// ---- XTS/Xpu/fb_Xpu.TcPOU
//---------------------------------------------------------------------------------------------------------------
//
//  HAUD 2023.12.14
//
//  - XTS_TRANSPORT_LAYER
//
//  fb_Xpu
//  - connect XTS_Utility.lib to TcCom
//  - cyclic plausibility checks
//  - cyclic ModuleInfoData
//
//  - connection to TcCom Server for local FB instances
//
//
//  CTRL / STATE --> see proprerties
//  structs for use of function block via mapping
//  cyclic check for new command
//
//  VAR INPUT / OUTPUT --> see properties
//
//---------------------------------------------------------------------------------------------------------------
// This SOFTWARE is provided as an Exemple by THE PROVIDER "as is" and "with all faults." THE PROVIDER makes no 
// representations or warranties of any kind concerning the safety, suitability, lack of viruses, inaccuracies, 
// typographical errors, or other harmful components of this SOFTWARE. There are inherent dangers in the use of 
// any software, and you are solely responsible for determining whether this SOFTWARE is compatible with your 
// equipment and other software installed on your equipment. You are also solely responsible for the protection 
// of your equipment and backup of your data, and THE PROVIDER will not be liable for any damages you may suffer 
// in connection with using, modifying, or distributing this SOFTWARE.
//---------------------------------------------------------------------------------------------------------------
FUNCTION_BLOCK fb_Xpu //IMPLEMENTS I_Xpu
VAR
  _eCheck                     : E_XPU_CHECK;
  _eInit                      : E_XPU_INIT;       // MUST equal INIT_DONE for anything to work
  _sVersionXpu                : STRING(80);       // only valid after successful init
  _sVersionNctController      : STRING(80);       // only valid afetr successful init
  //-------------------------------------------------------------------------------------------------
  // XTS Environment; ProcessingUnit, Part, Track, Mover
  //  - instances are initialized by getting OTCIDs
  //-------------------------------------------------------------------------------------------------
  _nXpu                       : UINT := 1;  // input property in case of multiple XPU in project
  _nGroup                     : UINT;       // input property in case of multiple Xpu in project

  _nTrack                     : UINT := 1;  // this example is intended for one track only

  {attribute 'displaymode':='hex'}
  _CaGroupOID                 : OTCID; // input property frome cyclic CA group interface, MUST be set in order to do successful INIT

  // checked and evaluated in XpuCheckCycle()
  _bAllPositionsValid,
  _bMoverIdDetectionValid,
  _bMoverIdDetectionError     : BOOL;

  _nDetectedMoverCount,
  _nExpectedMoverCount        : UINT;

  _XpuOperationMode           : OperationMode;
  _MoverIdDetectionMode       : MoverIdDetectionMode;

  // XTS_Utility connection to TcCOM Object
  _fbEnvironment              : Tc3_XTS_Utility.FB_TcIoXtsEnvironment;

  // local instances of members of Environment
  // local members are connected to TcCOM by XpuInit()
  _fbProcessingUnit           : Tc3_XTS_Utility.FB_TcIoXtsProcessingUnit;

  _fbXpuPart                  : Tc3_XTS_Utility.FB_TcIoXtsXpuPart;
  _fbXpuTrack                 : Tc3_XTS_Utility.FB_TcIoXtsXpuTrack;

  _fbMc2CaGroup               : Tc3_XTS_Utility.FB_Mc2CaGroup;

  _fbPartModules              : ARRAY[1..MAX_MODULE]  OF Tc3_XTS_Utility.FB_TcIoXtsPartModule;
  _fbMoverXpu                 : ARRAY[1..MAX_MOVER]   OF Tc3_XTS_Utility.FB_TcIoXtsXpuMover;

  _fbParameterSet             : ARRAY[1..MAX_PARAMETER_SET] OF Tc3_XTS_Utility.FB_TcIoXtsParameterSet;

  _fbNctController            : Tc3_XTS_Utility.FB_TcIoXtsNctController;

  _ItfNctBaseUnit              : ARRAY[1..MAX_NCT_BASE_UNIT] OF Tc3_XTS_Utility.I_TcIoXtsNctBaseUnitInterface;


  // TcCOM ObjectId (who am I talking to?)
  {attribute 'displaymode':='hex'}
  _Xpu_OTCID                  : OTCID;
  {attribute 'displaymode':='hex'}
  _Nct_OTCID                  : OTCID;
  {attribute 'displaymode':='hex'}
  _Group_OTCID                : ARRAY[1..MAX_GROUP]         OF OTCID; // OTCID read from XPU
  {attribute 'displaymode':='hex'}
  _Part_OTCID                 : ARRAY[1..MAX_PART]          OF OTCID;
  {attribute 'displaymode':='hex'}
  _Track_OTCID                : ARRAY[1..MAX_TRACK]         OF OTCID;
  {attribute 'displaymode':='hex'}
  _Mov_OTCID                  : ARRAY[1..MAX_MOVER]         OF OTCID;
  {attribute 'displaymode':='hex'}
  _Module_OTCID               : ARRAY[1..MAX_MODULE]        OF OTCID;
  {attribute 'displaymode':='hex'}
  _ParameterSet_OTCID         : ARRAY[1..MAX_PARAMETER_SET] OF OTCID;
  {attribute 'displaymode':='hex'}
  _NctBaseUnit_OTCID          : ARRAY[1..MAX_NCT_BASE_UNIT] OF OTCID;

  // COE Data access
  _ModuleInfoData             : REFERENCE TO ARRAY[1..MAX_MODULE] OF Tc3_XTS_Utility.ST_InfoDataView;
  _bModulePower               : ARRAY[1..MAX_MODULE] OF BOOL;

  // double check RailLength, XpuInit() will get stuck in error if not configured correctly
  _RailLengthXpu              : LREAL;
  _RailLengthGroup            : LREAL;

  _nLengthXpu,
  _nLengthGroup               : UINT;

  _nNctBaseUnitCount,
  _nParameterSetCount,
  _nInfoServerCount,
  _nIfoStationCount,
  _nPartCount,
  _nTrackCount,
  _nTaskCount,
  _nMoverCount,
  _nModuleCount               : UINT;

  _ix                         : UINT;

  {attribute 'hide'}
  _XpuInfo                    : ST_XPU_INFO;

  _stMsg                      : ST_Message;
  _eMessageLevel              : E_MessageType;
END_VAR

// get DcLink information from motor modules
PROPERTY AllModulesDcLink : bool
GET
VAR
  _bTmp     : BOOL;
  _nModule  : UINT;
END_VAR
IF NOT (_eInit = E_XPU_INIT.INIT_DONE) THEN RETURN; END_IF

FOR _nModule := 1 TO _nModuleCount
DO
  IF NOT _bModulePower[_nModule] // information comes from cyclic call in Cycle(): ModuleInfoData()
  THEN
    _bTmp  := FALSE;
    EXIT;
  ELSE
    _bTmp  := TRUE;
  END_IF
END_FOR

AllModulesDcLink := _bTmp;
END_GET
END_PROPERTY

PROPERTY CaGroupOID : OTCID
SET
// Group OTCID must come from the CA Group mapping in NC.Objects
_CaGroupOID := CaGroupOID;
END_SET
END_PROPERTY

METHOD Cycle : E_PROGRESS
VAR_INPUT
  Enable      : BOOL; // enable to do cyclic checks on Environment and its members
END_VAR
VAR_IN_OUT
  _eChk       : E_XPU_CHECK;
END_VAR
VAR_INST

  _eJobResult,
  _eResult      : E_PROGRESS;
  _eState       : E_PROGRESS := E_PROGRESS.PROGRESS_INIT;

END_VAR
IF NOT Enable
THEN
  ModuleInfoData(FALSE);

  _eResult  :=
  _eState   := E_PROGRESS.PROGRESS_INIT; 
  _eChk     := E_XPU_CHECK.INIT_CHECK;
END_IF 
//-----------------------------------------------------------------------------
// cyclic data fetch from Environment, ProcessingUnit, Part, ...
//-----------------------------------------------------------------------------
CASE _eState
OF
  E_PROGRESS.PROGRESS_INIT:
    IF Enable
    THEN
      _eState := _eResult         := E_PROGRESS.PROGRESS_BUSY;
    END_IF

  //---------------------------------------------------------------------------
  E_PROGRESS.PROGRESS_BUSY:       // get data from Xpu, ProcessingUnit, Part, XpuCaGroup
    _eState                       := E_PROGRESS.PROGRESS_STARTUP;

    _bAllPositionsValid           := _fbProcessingUnit.GetAreAllPositionsValid();
    _nDetectedMoverCount          := TO_UINT(_fbProcessingUnit.GetDetectedMoverCount());
    _nExpectedMoverCount          := TO_UINT(_fbProcessingUnit.GetExpectedMoverCount());
  
    _XpuOperationMode             := _fbProcessingUnit.GetOperationMode();
    _MoverIdDetectionMode         := _fbProcessingUnit.GetMoverIdDetectionMode();
  
    _RailLengthXpu                := _fbXpuPart.GetLength();
    _RailLengthGroup              := _fbMc2CaGroup.GetRailLength();
    _nLengthXpu                   := TO_UINT(_RailLengthXpu);
    _nLengthGroup                 := TO_UINT(_RailLengthGroup);
END_CASE
//-----------------------------------------------------------------------------
//-----------------------------------------------------------------------------
CASE _eState
OF
  //---------------------------------------------------------------------------
  E_PROGRESS.PROGRESS_STARTUP:    // check data for errors
    IF NOT (_bAllPositionsValid)
    THEN
      _eChk                       := E_XPU_CHECK.PROCESSING_UNIT_POSITIONS_VALID;
      _eState := _eResult         := E_PROGRESS.PROGRESS_ERROR;

      _stMsg.eType                := E_MessageType.eMessageError;
      _stMsg.eSubdevice           := e_Subdevice.Xpu_fbProcessingUnit;
      _stMsg.iErrorNumber         := 0;
      _stMsg.sText                := concat(TO_STRING(E_XPU_CHECK.PROCESSING_UNIT_POSITIONS_VALID), ': ');
      _stMsg.sText                := concat(_stMsg.sText, TO_STRING(_eResult));
      f_MessageSet(_stMsg);

    ELSIF NOT (_nLengthXpu > 0)
    THEN
      _eChk                       := E_XPU_CHECK.XPU_RAIL_LENGTH;
      _eState := _eResult         := E_PROGRESS.PROGRESS_ERROR;

      _stMsg.eType                := E_MessageType.eMessageError;
      _stMsg.eSubdevice           := e_Subdevice.Xpu_fbProcessingUnit;
      _stMsg.iErrorNumber         := 0;
      _stMsg.sText                := concat(TO_STRING(E_XPU_CHECK.XPU_RAIL_LENGTH), ': ');
      _stMsg.sText                := concat(_stMsg.sText, TO_STRING(_eResult));
      f_MessageSet(_stMsg);

    ELSIF NOT (_nLengthGroup > 0)
    THEN
      _eChk                       := E_XPU_CHECK.GROUP_RAIL_LENGTH;
      _eState := _eResult         := E_PROGRESS.PROGRESS_ERROR;
     
      _stMsg.eType                := E_MessageType.eMessageError;
      _stMsg.eSubdevice           := e_Subdevice.Xpu_fbProcessingUnit;
      _stMsg.iErrorNumber         := 0;
      _stMsg.sText                := concat(TO_STRING(E_XPU_CHECK.GROUP_RAIL_LENGTH), ': ');
      _stMsg.sText                := concat(_stMsg.sText, TO_STRING(_eResult));
      f_MessageSet(_stMsg);

    ELSIF NOT (_nDetectedMoverCount = _nExpectedMoverCount)
    THEN
      _bMoverIdDetectionValid     := FALSE;
      _eChk                       := E_XPU_CHECK.MOVER_COUNT_NOT_EQUAL;
      _eState := _eResult         := E_PROGRESS.PROGRESS_ERROR;

      _stMsg.eType                := E_MessageType.eMessageError;
      _stMsg.eSubdevice           := e_Subdevice.Xpu_fbProcessingUnit;
      _stMsg.iErrorNumber         := 0;
      _stMsg.sText                := concat(TO_STRING(E_XPU_CHECK.MOVER_COUNT_NOT_EQUAL), ': ');
      _stMsg.sText                := concat(_stMsg.sText, TO_STRING(_eResult));
      f_MessageSet(_stMsg);
  
    ELSIF NOT (_nLengthXpu = _nLengthGroup)
    THEN
      _eChk                       := E_XPU_CHECK.RAIL_LENGTH_COMPARE;
      _eState := _eResult         := E_PROGRESS.PROGRESS_ERROR;
 
      _stMsg.eType                := E_MessageType.eMessageError;
      _stMsg.eSubdevice           := e_Subdevice.Xpu_fbProcessingUnit;
      _stMsg.iErrorNumber         := 0;
      _stMsg.sText                := concat(TO_STRING(E_XPU_CHECK.RAIL_LENGTH_COMPARE), ': ');
      _stMsg.sText                := concat(_stMsg.sText, TO_STRING(_eResult));
      f_MessageSet(_stMsg);

    ELSE
      _eResult                    := E_PROGRESS.PROGRESS_WORKING;

      IF NOT (__ISVALIDREF(_ModuleInfoData))
      THEN
        _eState                   := E_PROGRESS.PROGRESS_BUSY;

        _stMsg.eType              := E_MessageType.eMessageError;
        _stMsg.eSubdevice         := e_Subdevice.Xpu_fbPartModules;
        _stMsg.iErrorNumber       := 0;
        _stMsg.sText              := concat(TO_STRING(_eState), ': ');
        _stMsg.sText              := concat(_stMsg.sText, 'NOT VALID _ModuleInfoData ref');
      ELSE
        _eJobResult               := ModuleInfoData(TRUE);
  
        IF (_eJobResult = E_PROGRESS.PROGRESS_DONE)
        THEN
          _eState                 := E_PROGRESS.PROGRESS_BUSY;
        END_IF  
      END_IF
    END_IF
END_CASE

Cycle                             := _eResult;
END_METHOD

METHOD GetEnvironment : I_TcIoXtsEnvironment
VAR_INPUT
END_VAR
IF NOT (_eInit = E_XPU_INIT.INIT_DONE) THEN RETURN; END_IF

GetEnvironment := _fbEnvironment;
END_METHOD

METHOD GetNctBaseUnit : Tc3_XTS_Utility.I_TcIoXtsNctBaseUnitInterface
VAR_INPUT
  Index     : UINT;
END_VAR
IF NOT (_eInit = E_XPU_INIT.INIT_DONE) THEN RETURN; END_IF

IF NOT (Index > 0) OR
   NOT (Index < MAX_NCT_BASE_UNIT+1)
THEN
  RETURN;
ELSE
  GetNctBaseUnit    := _ItfNctBaseUnit[Index];
END_IF
END_METHOD

METHOD GetNctController : Tc3_XTS_Utility.I_TcIoXtsNctController
VAR_INPUT
END_VAR
IF NOT (_eInit = E_XPU_INIT.INIT_DONE) THEN RETURN; END_IF

GetNctController := _fbNctController;
END_METHOD

METHOD GetParameterSet : I_TcIoXtsParameterSet
VAR_INPUT
  Index     : UINT;
END_VAR
IF NOT (_eInit = E_XPU_INIT.INIT_DONE) THEN RETURN; END_IF

IF NOT (Index > 0) OR
   NOT (Index < MAX_PARAMETER_SET+1)
THEN
  RETURN;
ELSE
  GetParameterSet   := _fbParameterSet[Index];
END_IF
END_METHOD

METHOD GetProcessingUnit : Tc3_XTS_Utility.I_TcIoXtsProcessingUnit
VAR_INPUT
END_VAR
IF NOT (_eInit = E_XPU_INIT.INIT_DONE) THEN RETURN; END_IF

GetProcessingUnit := _fbProcessingUnit;
END_METHOD

METHOD GetXpuMover : Tc3_XTS_Utility.I_TcIoXtsXpuMover
VAR_INPUT
  Index     : UINT;
END_VAR
IF NOT (_eInit = E_XPU_INIT.INIT_DONE) THEN RETURN; END_IF

IF NOT (Index > 0) OR
   NOT (Index < MAX_MOVER+1)
THEN
  RETURN;
ELSE
  GetXpuMover   := _fbMoverXpu[Index];
END_IF
END_METHOD

// mothers' little helper for display in visu
METHOD IdDetectionModeToString : string(20)
VAR
  _DetectionMode    : MoverIdDetectionMode; // Mover ID detection procedure
END_VAR
// just a little helper for visu display
IF NOT (_eInit = E_XPU_INIT.INIT_DONE) THEN IdDetectionModeToString := 'INIT required'; RETURN; END_IF

_DetectionMode := _fbProcessingUnit.GetMoverIdDetectionMode();

CASE _DetectionMode
OF
  MoverIdDetectionMode.Standard:
    IdDetectionModeToString       := 'Standard';

  MoverIdDetectionMode.Mover1:
    IdDetectionModeToString       := 'Mover 1';

  MoverIdDetectionMode.MultipleMover1:
    IdDetectionModeToString       := 'Multiple Mover 1';

ELSE
    IdDetectionModeToString       := 'UNKNOWN Mode';
END_CASE
END_METHOD

PROPERTY MessageLevel : e_messagetype
SET
_eMessageLevel := MessageLevel;
END_SET
END_PROPERTY

// mothers' little helper for display in visu
METHOD PRIVATE ModuleInfoData : E_PROGRESS
VAR_INPUT
  Enable        : BOOL; // enable to read ST_InfoDataView for diag/display
END_VAR
VAR_INST
  _idt,
  _nModule : UINT;
  _eReturn,
  _eState       : E_PROGRESS;
  _aPcbTemp     : ARRAY[1..4] OF REAL;
END_VAR
//---------------------------------------------------------------------------------------------
// just a little helper for visu display
// collects module data for local data
//---------------------------------------------------------------------------------------------
IF NOT (_eInit = E_XPU_INIT.INIT_DONE)      // if Xpu init is not done, just leave
THEN 
  RETURN; 
END_IF
//---------------------------------------------------------------------------------------------
IF NOT Enable                               // clear states on request
THEN
  _eReturn                                  := 
  _eState                                   := E_PROGRESS.PROGRESS_INIT; 
END_IF 
//---------------------------------------------------------------------------------------------
IF NOT (__ISVALIDREF(_ModuleInfoData))      // datafield not connected, error and leave
THEN
  ModuleInfoData                            := E_PROGRESS.PROGRESS_ERROR;
  RETURN;
END_IF
//---------------------------------------------------------------------------------------------
CASE _eState                                // get InfoData from motor modules
OF
  //-------------------------------------------------------------------------------------------
  E_PROGRESS.PROGRESS_INIT:
    IF Enable
    THEN
      _eState                                             := E_PROGRESS.PROGRESS_BUSY;
      _nModule                                            := 1;
    END_IF
END_CASE
CASE _eState
OF
  //-------------------------------------------------------------------------------------------
  E_PROGRESS.PROGRESS_BUSY:
    _eState                                               := E_PROGRESS.PROGRESS_PREPARE;

    _ModuleInfoData[_nModule].fAuxiliaryVoltage_5V        := _fbPartModules[_nModule].GetAuxiliaryVoltage5V();
    _ModuleInfoData[_nModule].fAuxiliaryVoltage_10V       := _fbPartModules[_nModule].GetAuxiliaryVoltage10V();
    _ModuleInfoData[_nModule].fAuxiliaryVoltage_24V       := _fbPartModules[_nModule].GetAuxiliaryVoltage24V();

    _ModuleInfoData[_nModule].fDcLinkVoltage              := _fbPartModules[_nModule].GetDCLinkVoltage();

    IF (_ModuleInfoData[_nModule].fDcLinkVoltage > 48.0*0.85) AND
       (_ModuleInfoData[_nModule].fDcLinkVoltage < 48.0*1.15)
    THEN
      _bModulePower[_nModule]                             := TRUE;
    ELSE
      _bModulePower[_nModule]                             := SEL((_XpuOperationMode = OperationMode.Simulation), FALSE, TRUE);
    END_IF

    _ModuleInfoData[_nModule].nCurrentScaling             := TO_INT(_fbPartModules[_nModule].GetCurrentScaling());

    _ModuleInfoData[_nModule].nDeviceInfo                 := _fbPartModules[_nModule].GetDeviceInfo();

    IF (_XpuOperationMode = OperationMode.Normal)
    THEN
      _ModuleInfoData[_nModule].fAverageTemp              := 0.0;
  
      _aPcbTemp                                           := _fbPartModules[_nModule].GetPCBTemperatures();
  
      _ModuleInfoData[_nModule].fPcbTemp_0                := _aPcbTemp[1];
      _ModuleInfoData[_nModule].fPcbTemp_1                := _aPcbTemp[2];
      _ModuleInfoData[_nModule].fPcbTemp_2                := _aPcbTemp[3];
      _ModuleInfoData[_nModule].fPcbTemp_3                := _aPcbTemp[4];

      FOR _idt := 1 TO 4
      DO
        _ModuleInfoData[_nModule].fAverageTemp            := _ModuleInfoData[_nModule].fAverageTemp + _aPcbTemp[_idt];
      END_FOR
      _ModuleInfoData[_nModule].fAverageTemp              := _ModuleInfoData[_nModule].fAverageTemp / 4;
    END_IF

    _ModuleInfoData[_nModule].fOverallCurrent             := _fbPartModules[_nModule].GetOverallCurrent();

    _ModuleInfoData[_nModule].fMaxDCLinkVoltageLast500ms  := _fbPartModules[_nModule].GetMaxDCLinkVoltageLast500ms();
    _ModuleInfoData[_nModule].fMaxOverallCurrentLast500ms := _fbPartModules[_nModule].GetMaxOverallCurrentLast500ms();
END_CASE
CASE _eState 
OF
  //-------------------------------------------------------------------------------------------
  E_PROGRESS.PROGRESS_PREPARE:
    IF (_nModule > _nModuleCount-1)
    THEN
      _eState                                             := E_PROGRESS.PROGRESS_WORKING;
    ELSE
      _nModule                                            := _nModule + 1;
      _eReturn                                            :=
      _eState                                             := E_PROGRESS.PROGRESS_BUSY;
    END_IF

  //-------------------------------------------------------------------------------------------
  E_PROGRESS.PROGRESS_WORKING:
    _eReturn                                              := E_PROGRESS.PROGRESS_DONE;
    _eState                                               := E_PROGRESS.PROGRESS_INIT;
END_CASE

ModuleInfoData                                            := _eReturn;
END_METHOD

// mothers' little helper for display in visu
METHOD MoverPositionAssignementToString : string(20)
VAR
  _PositionAssignement    : MoverPositionAssignment; // XPU movver assignement procedure
END_VAR
// just a little helper for visu display
IF NOT (_eInit = E_XPU_INIT.INIT_DONE) THEN MoverPositionAssignementToString := 'INIT required'; RETURN; END_IF

_PositionAssignement      := _fbProcessingUnit.GetMoverPositionAssignment();

CASE _PositionAssignement
OF
  MoverPositionAssignment.Standard:
    MoverPositionAssignementToString    := 'Standard';

  MoverPositionAssignment.StartAtFirstMover:
    MoverPositionAssignementToString    := 'Start At First Mover';
ELSE
    MoverPositionAssignementToString    := 'UNKNOWN Assgnement';
END_CASE
END_METHOD

// mothers' little helper for display in visu
METHOD OpModeToString : String(20)
VAR
  _OpMode     : OperationMode; // XPU operation mode
END_VAR
// just a little helper for visu display
IF NOT (_eInit = E_XPU_INIT.INIT_DONE) THEN OpModeToString := 'INIT required'; RETURN; END_IF

_OpMode   := _fbProcessingUnit.GetOperationMode();

CASE _OpMode
OF
  OperationMode.Normal:
    OpModeToString      := 'Normal';

  OperationMode.Simulation:
    OpModeToString      := 'Simulation';

ELSE
    OpModeToString      := 'UNKNOWN OP MODE';
END_CASE
END_METHOD

PROPERTY RailLength : lreal
GET
IF (_eInit = E_XPU_INIT.INIT_DONE)
THEN
  RailLength := _fbXpuPart.GetLength();
ELSE
  RailLength := 0.0;
END_IF
END_GET
END_PROPERTY

PROPERTY XpuInfo : st_xpu_info
GET
IF NOT (_eInit = E_XPU_INIT.INIT_DONE) THEN RETURN; END_IF

_XpuInfo.AllPositionsValid        := _bAllPositionsValid;

_XpuInfo.IdDetectionError         := _bMoverIdDetectionError;
_XpuInfo.IdDetectionValid         := _bMoverIdDetectionValid;

_XpuInfo.IdDetectionActive        := _fbProcessingUnit.GetIsMoverIdDetectionActive();

_XpuInfo.OperationMode            := TO_UINT(_fbProcessingUnit.GetOperationMode());

_XpuInfo.IdDetectionMode          := TO_UINT(_fbProcessingUnit.GetMoverIdDetectionMode());
_XpuInfo.MoverPositionAssignement := TO_UINT(_fbProcessingUnit.GetMoverPositionAssignment());

_XpuInfo.nDetectedAxisCount       := _nDetectedMoverCount;
_XpuInfo.nExpectedAxisCount       := _nExpectedMoverCount;

_XpuInfo.nParameterSetCount       := _nParameterSetCount;

XpuInfo := _XpuInfo;
END_GET
END_PROPERTY

METHOD PROTECTED XpuInit  : E_XPU_INIT      // connect to TcCOM
VAR_INPUT
  Execute       : BOOL;           // must be executed for connecting to TcCOM Environment of Xpu
END_VAR
VAR_IN_OUT
  _eReslt       : E_PROGRESS;     // send info about progress to caller
  _eChk         : E_XPU_CHECK;
END_VAR
VAR_INST
  _eState           : E_PROGRESS;   // progress state
  _nState           : E_XPU_INIT;   // initialization state
  _eDataGetCount    : E_PROGRESS;   // cycle counter to catch exceeding wait time for data from ProcessingUnit

  _nParaSetIdx      : UINT;

  _nMoverIdx,
  _nModuleIdx       : UINT;

  _nNctBaseUnitIdx        : UINT;
END_VAR
//-----------------------------------------------------------------------------------------------
//-----------------------------------------------------------------------------------------------
// clear progress on request
IF NOT Execute 
THEN 
  _eState                           := E_PROGRESS.PROGRESS_INIT;
  _eDataGetCount                    := 0;
 
  XpuInit                           :=
  _nState                           := E_XPU_INIT.INIT_START; 
  RETURN; 
END_IF
//-----------------------------------------------------------------------------------------------
//-----------------------------------------------------------------------------------------------
// progress state
//-----------------------------------------------------------------------------------------------
//-----------------------------------------------------------------------------------------------
CASE _eState
OF
  E_PROGRESS.PROGRESS_INIT:         // clear start
    IF Execute
    THEN
      _eState                       := E_PROGRESS.PROGRESS_BUSY;
      _eChk                         := E_XPU_CHECK.INIT_CHECK;    // clear cyclic check state
      _sVersionNctController        :=
      _sVersionXpu                  := TO_STRING(_eChk);          // clear Version string

      // always initialize environment function blocks to get defined start of progress
      _fbEnvironment.Init(FALSE);
      _fbEnvironment.GetXpuOids(FALSE);
      _fbEnvironment.GetInfoServerOids(FALSE);

      // clear initialization states
      _nState                       := E_XPU_INIT.INIT_START;

      // clear check bits
      _bAllPositionsValid           :=
      _bMoverIdDetectionValid       :=
      _bMoverIdDetectionError       := FALSE;

      // clear check values
      _nLengthXpu                   :=
      _nLengthGroup                 :=
      _nDetectedMoverCount          :=
      _nExpectedMoverCount          := 0;

      // clear work values
      _nNctBaseUnitCount            :=
      _nNctBaseUnitIdx              :=
      _nParameterSetCount           :=
      _nInfoServerCount             :=
      _nIfoStationCount             :=
      _nPartCount                   :=
      _nTrackCount                  :=
      _nTaskCount                   :=
      _nMoverCount                  :=
      _nModuleCount                 :=
      _nMoverIdx                    :=
      _nModuleIdx                   := 0;

      IF (_eMessageLevel = E_MessageType.eMessageVerbose)
      THEN
        _stMsg.eType                := E_MessageType.eMessageVerbose;
        _stMsg.eSubdevice           := e_Subdevice.Xpu_fbEnvironment;
        _stMsg.iErrorNumber         := 0;
        _stMsg.sText                := concat(TO_STRING(_eState), ': ');
        _stMsg.sText                := concat(_stMsg.sText, TO_STRING(_eChk));
        f_MessageSet(_stMsg);
      END_IF
    END_IF
END_CASE
//-----------------------------------------------------------------------------------------------
//-----------------------------------------------------------------------------------------------
//-----------------------------------------------------------------------------------------------
CASE _eState
OF
  E_PROGRESS.PROGRESS_BUSY:         // begin with initializing environment
    CASE _nState
    OF
  //-----------------------------------------------------------------------------------------------
  //-----------------------------------------------------------------------------------------------
  INIT_START:                       // call initialization of environment

    IF NOT _fbEnvironment.P_IsInitialized
    THEN
      _fbEnvironment.Init(TRUE);
    END_IF

    IF (_fbEnvironment.bError)
    THEN
      _eChk                         := E_XPU_CHECK.INIT_CHECK_ERROR;
                                    
      _stMsg.eType                  := E_MessageType.eMessageError;
      _stMsg.eSubdevice             := e_Subdevice.Xpu_fbEnvironment;
      _stMsg.iErrorNumber           := 666;
      _stMsg.sText                  := concat(TO_STRING(_eState), ': ');
      _stMsg.sText                  := concat(_stMsg.sText, TO_STRING(_eChk));
      f_MessageSet(_stMsg);

      _eState                       := E_PROGRESS.PROGRESS_ERROR;

    // get information about success in Property (P_<function>)
    ELSIF _fbEnvironment.P_IsInitialized
    THEN
      // now environment is initialized
     
      //---------------------------------------------------------------------
      // use of local function block instances
      // get information about Object IDs to local datafields
      //---------------------------------------------------------------------
      //  - everything else in this state machine is for use within fb_Xpu
      //  - the following states shall illustrate how TcCOM Objects are connected through XTS_Utility lib
      //  - local instances of members of Environment are connected from here onward
      //
      IF _fbEnvironment.GetXpuOids(TRUE) // get object IDs for all processing units
      THEN
        _fbEnvironment.Init(FALSE);// clear environment init
        _nState                     := INIT_ENVIRONMENT_OID;

        IF (_eMessageLevel = E_MessageType.eMessageVerbose)
        THEN
          _stMsg.eType              := E_MessageType.eMessageVerbose;
          _stMsg.eSubdevice         := e_Subdevice.Xpu_fbEnvironment;
          _stMsg.iErrorNumber       := 0;
          _stMsg.sText              := concat(TO_STRING(_eState), ': ');
          _stMsg.sText              := concat(_stMsg.sText, TO_STRING(_nState));
          f_MessageSet(_stMsg);
        END_IF
      END_IF
    END_IF

  //-----------------------------------------------------------------------------------------------
  //-----------------------------------------------------------------------------------------------
  INIT_ENVIRONMENT_OID:             // get processing unit object ID for THIS instance
    _Xpu_OTCID                      := _fbEnvironment.P_XpuOids[_nXpu];   // fb_Xpu.XpuInstance --> _nXpu

    // clear all local object IDs
    memset(ADR(_Part_OTCID)         , 0, SIZEOF(_Part_OTCID));
    memset(ADR(_Track_OTCID)        , 0, SIZEOF(_Track_OTCID));
    memset(ADR(_Mov_OTCID)          , 0, SIZEOF(_Mov_OTCID));
    memset(ADR(_Module_OTCID)       , 0, SIZEOF(_Module_OTCID));
    memset(ADR(_ParameterSet_OTCID) , 0, SIZEOF(_ParameterSet_OTCID));

    // clear function blocks
    _fbEnvironment.GetXpuOids           (FALSE);
    _fbEnvironment.GetCaGroupCount      (FALSE);
    _fbEnvironment.GetInfoServerCount   (FALSE);
    _fbEnvironment.GetParameterSetCount (FALSE);

    _eState                         := E_PROGRESS.PROGRESS_PREPARE; // TODO - implement InfoServer R/W
    _nState                         := INIT_CA_GROUP_OID;           // TODO - implement initialization states for info server procedure

    //_nState                       := INIT_INFO_SERVER_ITF;              // check environment for info servers

  //-----------------------------------------------------------------------------------------------
  //-----------------------------------------------------------------------------------------------
  INIT_INFO_SERVER_ITF:           // HAUD 2024 03 14: TODO - implement procedure for getting Info server data to local datafields
    IF _fbEnvironment.GetInfoServerCount(TRUE)
    THEN
      // how many of you are there?
      _nInfoServerCount             := _fbEnvironment.P_InfoServerCount;

      IF (_nInfoServerCount > 0)
      THEN
        // go do something with the data
        //
        //  TODO - get station coordinates
        _eState                     := E_PROGRESS.PROGRESS_PREPARE; // TODO - implement InfoServer R/W
        _nState                     := INIT_CA_GROUP_OID;           // TODO - implement initialization states for info server procedure

        IF (_eMessageLevel = E_MessageType.eMessageVerbose)
        THEN
          _stMsg.eType              := E_MessageType.eMessageVerbose;
          _stMsg.eSubdevice         := e_Subdevice.Xpu_fbEnvironment;
          _stMsg.iErrorNumber       := 0;
          _stMsg.sText              := concat(TO_STRING(_eState), ': ');
          _stMsg.sText              := concat(_stMsg.sText, TO_STRING(_nState));
          f_MessageSet(_stMsg);
        END_IF

      ELSE
        // no info server present
        _eState                     := E_PROGRESS.PROGRESS_PREPARE;
        _nState                     := INIT_CA_GROUP_OID; // go check CA group

        IF (_eMessageLevel = E_MessageType.eMessageVerbose)
        THEN
          _stMsg.eType              := E_MessageType.eMessageVerbose;
          _stMsg.eSubdevice         := e_Subdevice.Xpu_fbEnvironment;
          _stMsg.iErrorNumber       := 0;
          _stMsg.sText              := concat(TO_STRING(_eState), ': ');
          _stMsg.sText              := concat(_stMsg.sText, TO_STRING(_nState));
          f_MessageSet(_stMsg);
        END_IF
      END_IF
    END_IF
  END_CASE
END_CASE
//-----------------------------------------------------------------------------------------------
//-----------------------------------------------------------------------------------------------
//-----------------------------------------------------------------------------------------------
CASE _eState
OF
  E_PROGRESS.PROGRESS_PREPARE:      // CA group initialization
  CASE _nState
  OF
  //-----------------------------------------------------------------------------------------------
  //-----------------------------------------------------------------------------------------------
  INIT_CA_GROUP_OID:                // get object IDs of all CA groups in environment
    IF _fbEnvironment.GetCaGroupOids(TRUE)
    THEN
      _Group_OTCID                  := _fbEnvironment.P_CaGroupOids;  // copy all Ids to local
      _nState                       := INIT_CA_GROUP_GET_OID;

      IF (_eMessageLevel = E_MessageType.eMessageVerbose)
      THEN
        _stMsg.eType                := E_MessageType.eMessageVerbose;
        _stMsg.eSubdevice           := e_Subdevice.Xpu_fbEnvironment;
        _stMsg.iErrorNumber         := 0;
        _stMsg.sText                := concat(TO_STRING(_eState), ': ');
        _stMsg.sText                := concat(_stMsg.sText, TO_STRING(_nState));
        f_MessageSet(_stMsg);
      END_IF
    END_IF

  //-----------------------------------------------------------------------------------------------
  //-----------------------------------------------------------------------------------------------
  INIT_CA_GROUP_GET_OID:            // look for any CA group
    _fbEnvironment.GetCaGroupOids(FALSE);
    IF NOT (_Group_OTCID[1] <> 0)
    THEN
      // no group is configured in project --> error, go add/link CA Group in NC objects
      _eChk                         := E_XPU_CHECK.GROUP_NOT_CONFIGURED;
      _eState                       := E_PROGRESS.PROGRESS_ERROR;

      _stMsg.eType                  := E_MessageType.eMessageError;
      _stMsg.eSubdevice             := e_Subdevice.Xpu_fbEnvironment;
      _stMsg.iErrorNumber           := 0;
      _stMsg.sText                  := concat(TO_STRING(_eState), ': ');
      _stMsg.sText                  := concat(_stMsg.sText, TO_STRING(_nState));
      f_MessageSet(_stMsg);
    ELSE
      _nState                       := INIT_CA_GROUP_CHECK_OID; // get matching CA group

      IF (_eMessageLevel = E_MessageType.eMessageVerbose)
      THEN
        _stMsg.eType                := E_MessageType.eMessageVerbose;
        _stMsg.eSubdevice           := e_Subdevice.Xpu_fbEnvironment;
        _stMsg.iErrorNumber         := 0;
        _stMsg.sText                := concat(TO_STRING(_eState), ': ');
        _stMsg.sText                := concat(_stMsg.sText, TO_STRING(_nState));
        //f_MessageSet(_stMsg);
      END_IF
    END_IF

  //-----------------------------------------------------------------------------------------------
  //-----------------------------------------------------------------------------------------------
  INIT_CA_GROUP_CHECK_OID:          // ID must be found, there is one chance
    _eChk                           := E_XPU_CHECK.GROUP_OID_MISMATCH;
    _eState                         := E_PROGRESS.PROGRESS_ERROR;

    FOR _ix := 1 TO MAX_GROUP
    DO
      IF (_fbEnvironment.P_CaGroupOids[_ix] <> 0)
      THEN
        // check whether the input from cyclic interface can be found in XPU data
        IF (_fbEnvironment.P_CaGroupOids[_ix] = _CaGroupOID)  // _CaGroupOID must be linked from NC Objects into PLC (GROUP_REF)
        THEN

          _eState                   := E_PROGRESS.PROGRESS_PREPARE; // stay here
          _eChk                     := E_XPU_CHECK.INIT_CHECK;

          _nGroup                   := _ix;

          _fbEnvironment.GetCaGroupOids(FALSE);
          _nState                   := INIT_CA_GROUP_COM; // only continue if match was found

          IF (_eMessageLevel = E_MessageType.eMessageVerbose)
          THEN
            _stMsg.eType            := E_MessageType.eMessageVerbose;
            _stMsg.eSubdevice       := e_Subdevice.Xpu_fbEnvironment;
            _stMsg.iErrorNumber     := _CaGroupOID;
            _stMsg.sText            := concat(TO_STRING(_eState), ': ');
            _stMsg.sText            := concat(_stMsg.sText, TO_STRING(_nState));
            f_MessageSet(_stMsg);
          END_IF
          EXIT;
        END_IF
      END_IF
    END_FOR

    IF (_eState = E_PROGRESS.PROGRESS_ERROR)
    THEN
      _stMsg.eType                  := E_MessageType.eMessageError;
      _stMsg.eSubdevice             := e_Subdevice.Xpu_fbEnvironment;
      _stMsg.iErrorNumber           := _nGroup;
      _stMsg.sText                  := concat(TO_STRING(_eState), ': ');
      _stMsg.sText                  := concat(_stMsg.sText, TO_STRING(_nState));
      f_MessageSet(_stMsg);
    END_IF

  //-----------------------------------------------------------------------------------------------
  //-----------------------------------------------------------------------------------------------
  INIT_CA_GROUP_COM:                // connect to CaGroup function block in environment
    IF (_fbMc2CaGroup.GetComObject(_fbEnvironment.P_CaGroupOids[_nGroup]))
    THEN
      _fbEnvironment.GetParameterSetCount(FALSE);

      _nState                       := INIT_PARAMETERSET_COUNT;

      IF (_eMessageLevel = E_MessageType.eMessageVerbose)
      THEN
        _stMsg.eType                := E_MessageType.eMessageVerbose;
        _stMsg.eSubdevice           := e_Subdevice.Xpu_fbEnvironment;
        _stMsg.iErrorNumber         := _nGroup;
        _stMsg.sText                := concat(TO_STRING(_eState), ': ');
        _stMsg.sText                := concat(_stMsg.sText, TO_STRING(_nState));
       f_MessageSet(_stMsg);
      END_IF
    END_IF

  //-----------------------------------------------------------------------------------------------
  //-----------------------------------------------------------------------------------------------
  INIT_PARAMETERSET_COUNT:
    IF _fbEnvironment.GetParameterSetCount(TRUE)
    THEN
      _fbEnvironment.GetParameterSetOids(FALSE);
      _nParaSetIdx                  :=
      _nParameterSetCount           := _fbEnvironment.P_ParameterSetCount;
      _nState                       := INIT_PARAMETERSET_OID; 

      IF (_eMessageLevel = E_MessageType.eMessageVerbose)
      THEN
        _stMsg.eType                := E_MessageType.eMessageVerbose;
        _stMsg.eSubdevice           := e_Subdevice.Xpu_fbEnvironment;
        _stMsg.iErrorNumber         := _nParameterSetCount;
        _stMsg.sText                := concat(TO_STRING(_eState), ': ');
        _stMsg.sText                := concat(_stMsg.sText, TO_STRING(_nState));
        f_MessageSet(_stMsg);
      END_IF
    END_IF

  //-----------------------------------------------------------------------------------------------
  //-----------------------------------------------------------------------------------------------
  INIT_PARAMETERSET_OID:
    IF (_nParameterSetCount = 0)
    THEN
      _fbEnvironment.GetParameterSetCount(FALSE);
      _eState                       := E_PROGRESS.PROGRESS_STARTUP;
      _nState                       := INIT_PROCESSING_UNIT_COM;

    ELSIF _fbEnvironment.GetParameterSetOids(TRUE)
    THEN
      _fbEnvironment.GetParameterSetCount(FALSE);
      _ParameterSet_OTCID           := _fbEnvironment.P_ParameterSetOids;
      _nState                       := INIT_PARAMETERSET_COM;
    END_IF

  //-----------------------------------------------------------------------------------------------
  //-----------------------------------------------------------------------------------------------
  INIT_PARAMETERSET_COM:
    IF (_nParaSetIdx > 0)
    THEN
      IF _fbParameterSet[_nParaSetIdx].GetComObject(_ParameterSet_OTCID[_nParaSetIdx])
      THEN
        _nState                     := INIT_PARAMETERSET_COM_NEXT;

        IF (_eMessageLevel = E_MessageType.eMessageVerbose)
        THEN
          _stMsg.eType              := E_MessageType.eMessageVerbose;
          _stMsg.eSubdevice         := e_Subdevice.Xpu_fbParameterSet;
          _stMsg.iErrorNumber       := _ParameterSet_OTCID[_nParaSetIdx];
          _stMsg.sText              := concat(TO_STRING(_eState), ': ');
          _stMsg.sText              := concat(_stMsg.sText, TO_STRING(_nState));
          f_MessageSet(_stMsg);
        END_IF
      END_IF
    ELSE
      _fbEnvironment.GetParameterSetOids(FALSE);
      _eState                       := E_PROGRESS.PROGRESS_STARTUP;
      _nState                       := INIT_PROCESSING_UNIT_COM;
    END_IF
      

  //-----------------------------------------------------------------------------------------------
  //-----------------------------------------------------------------------------------------------
  INIT_PARAMETERSET_COM_NEXT:
    _nParaSetIdx                    := _nParaSetIdx - 1;
    _nState                         := INIT_PARAMETERSET_COM; 
  END_CASE
END_CASE
//-----------------------------------------------------------------------------------------------
//-----------------------------------------------------------------------------------------------
//-----------------------------------------------------------------------------------------------
CASE _eState
OF
  E_PROGRESS.PROGRESS_STARTUP:      // ProcessingUnit initialization
  CASE _nState
  OF
  //-----------------------------------------------------------------------------------------------
  //-----------------------------------------------------------------------------------------------
  INIT_PROCESSING_UNIT_COM:         // connect local function block with TcCom object
    IF (_fbProcessingUnit.GetComObject(_Xpu_OTCID))
    THEN
      // local function block can now be used to get information
      // get operation mode first
      _XpuOperationMode             := _fbProcessingUnit.GetOperationMode();
      _nState                       := INIT_PROCESSING_UNIT_PART_COUNT;

      IF (_eMessageLevel = E_MessageType.eMessageVerbose)
      THEN
        _stMsg.eType                := E_MessageType.eMessageVerbose;
        _stMsg.eSubdevice           := e_Subdevice.Xpu_fbProcessingUnit;
        _stMsg.iErrorNumber         := _nGroup;
        _stMsg.sText                := concat(TO_STRING(_eState), ': ');
        _stMsg.sText                := concat(_stMsg.sText, TO_STRING(_nState));
        f_MessageSet(_stMsg);
      END_IF
    END_IF

  //-----------------------------------------------------------------------------------------------
  //-----------------------------------------------------------------------------------------------
  INIT_PROCESSING_UNIT_PART_COUNT:  // get parts in ProcessingUnit
    _nPartCount                     := TO_UINT(_fbProcessingUnit.GetPartCount());

    IF (_nPartCount > 0)            // one is enough
    THEN
      _nState                       := INIT_PROCESSING_UNIT_PART_OID;

      IF (_eMessageLevel = E_MessageType.eMessageVerbose)
      THEN
        _stMsg.eType                := E_MessageType.eMessageVerbose;
        _stMsg.eSubdevice           := e_Subdevice.Xpu_fbProcessingUnit;
        _stMsg.iErrorNumber         := _nGroup;
        _stMsg.sText                := concat(TO_STRING(_eState), ': ');
        _stMsg.sText                := concat(_stMsg.sText, TO_STRING(_nState));
        f_MessageSet(_stMsg);
      END_IF
    END_IF

  //-----------------------------------------------------------------------------------------------
  //-----------------------------------------------------------------------------------------------
  INIT_PROCESSING_UNIT_PART_OID:    // get object IDs of all parts in ProcessingUNit
    IF _fbProcessingUnit.GetPartOids()
    THEN
      _Part_OTCID                   := _fbProcessingUnit.P_PartOids;  // copy IDs to local
      _nState                       := INIT_PROCESSING_UNIT_TRACK_COUNT;

      IF (_eMessageLevel = E_MessageType.eMessageVerbose)
      THEN
        _stMsg.eType                := E_MessageType.eMessageVerbose;
        _stMsg.eSubdevice           := e_Subdevice.Xpu_fbProcessingUnit;
        _stMsg.iErrorNumber         := _nGroup;
        _stMsg.sText                := concat(TO_STRING(_eState), ': ');
        _stMsg.sText                := concat(_stMsg.sText, TO_STRING(_nState));
        f_MessageSet(_stMsg);
      END_IF
    END_IF

  //-----------------------------------------------------------------------------------------------
  //-----------------------------------------------------------------------------------------------
  INIT_PROCESSING_UNIT_TRACK_COUNT: // how many tracks does this ProcessingUnit have?
    _nTrackCount                    := TO_UINT(_fbProcessingUnit.GetTrackCount());
  
    IF (_nTrackCount > 0)           // one is enough
    THEN
      _nState                       := INIT_PROCESSING_UNIT_TRACK_OID;

      IF (_eMessageLevel = E_MessageType.eMessageVerbose)
      THEN
        _stMsg.eType                := E_MessageType.eMessageVerbose;
        _stMsg.eSubdevice           := e_Subdevice.Xpu_fbProcessingUnit;
        _stMsg.iErrorNumber         := _nTrackCount;
        _stMsg.sText                := concat(TO_STRING(_eState), ': ');
        _stMsg.sText                := concat(_stMsg.sText, TO_STRING(_nState));
        f_MessageSet(_stMsg);
      END_IF
    END_IF

  //-----------------------------------------------------------------------------------------------
  //-----------------------------------------------------------------------------------------------
  INIT_PROCESSING_UNIT_TRACK_OID:   // get object IDs of all tracks in ProcessingUnit
    IF _fbProcessingUnit.GetTrackOids()
    THEN
      _Track_OTCID                  := _fbProcessingUnit.P_TrackOids; // copy IDs to local
      _nState                       := INIT_PROCESSING_UNIT_MOVER_COUNT;

      IF (_eMessageLevel = E_MessageType.eMessageVerbose)
      THEN
        _stMsg.eType                := E_MessageType.eMessageVerbose;
        _stMsg.eSubdevice           := e_Subdevice.Xpu_fbProcessingUnit;
        _stMsg.iErrorNumber         := 0;
        _stMsg.sText                := concat(TO_STRING(_eState), ': ');
        _stMsg.sText                := concat(_stMsg.sText, TO_STRING(_nState));
        f_MessageSet(_stMsg);
      END_IF
    END_IF

  //-----------------------------------------------------------------------------------------------
  //-----------------------------------------------------------------------------------------------
  INIT_PROCESSING_UNIT_MOVER_COUNT: // how many of you are there?
    _nMoverCount                    := TO_UINT(_fbProcessingUnit.GetMoverCount());
  
    IF (_nMoverCount > 0)           // one is enough
    THEN
      _nState                       := INIT_PROCESSING_UNIT_MOVER_OID;

      IF (_eMessageLevel = E_MessageType.eMessageVerbose)
      THEN
        _stMsg.eType                := E_MessageType.eMessageVerbose;
        _stMsg.eSubdevice           := e_Subdevice.Xpu_fbProcessingUnit;
        _stMsg.iErrorNumber         := _nMoverCount;
        _stMsg.sText                := concat(TO_STRING(_eState), ': ');
        _stMsg.sText                := concat(_stMsg.sText, TO_STRING(_nState));
        f_MessageSet(_stMsg);
      END_IF
    END_IF

  //-----------------------------------------------------------------------------------------------
  //-----------------------------------------------------------------------------------------------
  INIT_PROCESSING_UNIT_MOVER_OID:   // get object IDs of all mover in ProcessingUnit
    IF _fbProcessingUnit.GetMoverOids()
    THEN
      _Mov_OTCID                    := _fbProcessingUnit.P_MoverOids; // copy IDs to local
      _nState                       := INIT_PROCESSING_UNIT_TASK_COUNT;
      _eChk                         := E_XPU_CHECK.MOVER_COUNT;

      IF (_eMessageLevel = E_MessageType.eMessageVerbose)
      THEN
        _stMsg.eType                := E_MessageType.eMessageVerbose;
        _stMsg.eSubdevice           := e_Subdevice.Xpu_fbProcessingUnit;
        _stMsg.iErrorNumber         := 0;
        _stMsg.sText                := concat(TO_STRING(_eState), ': ');
        _stMsg.sText                := concat(_stMsg.sText, TO_STRING(_nState));
        f_MessageSet(_stMsg);
      END_IF
    END_IF

  //-----------------------------------------------------------------------------------------------
  //-----------------------------------------------------------------------------------------------
  INIT_PROCESSING_UNIT_TASK_COUNT:  // how many?
    _nTaskCount                     := TO_UINT(_fbProcessingUnit.GetTaskCount());
  
    IF (_nTaskCount > 0)
    THEN
      _nState                       := INIT_PROCESSING_UNIT_TASK_OID;

      IF (_eMessageLevel = E_MessageType.eMessageVerbose)
      THEN
        _stMsg.eType                := E_MessageType.eMessageVerbose;
        _stMsg.eSubdevice           := e_Subdevice.Xpu_fbProcessingUnit;
        _stMsg.iErrorNumber         := _nTaskCount;
        _stMsg.sText                := concat(TO_STRING(_eState), ': ');
        _stMsg.sText                := concat(_stMsg.sText, TO_STRING(_nState));
        f_MessageSet(_stMsg);
      END_IF
    END_IF    

  //-----------------------------------------------------------------------------------------------
  //-----------------------------------------------------------------------------------------------
  INIT_PROCESSING_UNIT_TASK_OID:    // get their names!
    IF _fbProcessingUnit.GetTaskOids()
    THEN
      _eState                       := E_PROGRESS.PROGRESS_CHECK;
      _nState                       := INIT_NCT_CONTROLLER_OID;

      IF (_eMessageLevel = E_MessageType.eMessageVerbose)
      THEN
        _stMsg.eType                := E_MessageType.eMessageVerbose;
        _stMsg.eSubdevice           := e_Subdevice.Xpu_fbNctController;
        _stMsg.iErrorNumber         := _nTrack;
        _stMsg.sText                := concat(TO_STRING(_eState), ': ');
        _stMsg.sText                := concat(_stMsg.sText, TO_STRING(_nState));
        f_MessageSet(_stMsg);
      END_IF
    END_IF
  END_CASE
END_CASE
//-----------------------------------------------------------------------------------------------
//-----------------------------------------------------------------------------------------------
//-----------------------------------------------------------------------------------------------
CASE _eState
OF
  E_PROGRESS.PROGRESS_CHECK:        // NCT
  CASE _nState
  OF
  //-----------------------------------------------------------------------------------------------
  //-----------------------------------------------------------------------------------------------
  INIT_NCT_CONTROLLER_OID:
    IF (_fbProcessingUnit.GetNctControllerOid())
    THEN
      _Nct_OTCID                    := _fbProcessingUnit.P_NctControllerOid;

      IF NOT(_Nct_OTCID > 0)
      THEN
        _eState                     := E_PROGRESS.PROGRESS_OCCUPIED;
      ELSE
        _eState                     := E_PROGRESS.PROGRESS_CHECK;
        _nState                     := INIT_NCT_CONTROLLER_COM;

        IF (_eMessageLevel = E_MessageType.eMessageVerbose)
        THEN
          _stMsg.eType              := E_MessageType.eMessageVerbose;
          _stMsg.eSubdevice         := e_Subdevice.Xpu_fbNctController;
          _stMsg.iErrorNumber       := 0;
          _stMsg.sText              := concat(TO_STRING(_eState), ': ');
          _stMsg.sText              := concat(_stMsg.sText, TO_STRING(_nState));
          f_MessageSet(_stMsg);
        END_IF
      END_IF
    END_IF

  //-----------------------------------------------------------------------------------------------
  //-----------------------------------------------------------------------------------------------
  INIT_NCT_CONTROLLER_COM:
    IF (_fbNctController.GetComObject(_Nct_OTCID))
    THEN
      _sVersionNctController        := _fbNctController.GetVersionString();
      _nState                       := INIT_NCT_BASE_UNIT_COUNT;

      IF (_eMessageLevel = E_MessageType.eMessageVerbose)
      THEN
        _stMsg.eType                := E_MessageType.eMessageVerbose;
        _stMsg.eSubdevice           := e_Subdevice.Xpu_fbNctController;
        _stMsg.iErrorNumber         := 0;
        _stMsg.sText                := concat(TO_STRING(_eState), ': ');
        _stMsg.sText                := concat(_stMsg.sText, TO_STRING(_nState));
        f_MessageSet(_stMsg);
      END_IF
      IF (_eMessageLevel > E_MessageType.eMessageError)
      THEN
        _stMsg.eType                := E_MessageType.eMessageInfo;
        _stMsg.eSubdevice           := e_Subdevice.Xpu_fbNctController;
        _stMsg.iErrorNumber         := 0;
        _stMsg.sText                := concat('NctController VersionString: ', _sVersionNctController);
        f_MessageSet(_stMsg);
      END_IF
    END_IF

  //-----------------------------------------------------------------------------------------------
  //-----------------------------------------------------------------------------------------------
  INIT_NCT_BASE_UNIT_COUNT:
    _nNctBaseUnitCount              := TO_UINT(_fbNctController.GetBaseUnitInterfaceCount());

    IF NOT (_nNctBaseUnitCount > 0)
    THEN
      _eState                       := E_PROGRESS.PROGRESS_OCCUPIED;

      IF (_eMessageLevel = E_MessageType.eMessageVerbose)
      THEN
        _stMsg.eType                := E_MessageType.eMessageVerbose;
        _stMsg.eSubdevice           := e_Subdevice.Xpu_fbNctBaseUnit;
        _stMsg.iErrorNumber         := 0;
        _stMsg.sText                := concat(TO_STRING(_eState), ': ');
        _stMsg.sText                := concat(_stMsg.sText, TO_STRING(_nState));
        f_MessageSet(_stMsg);
      END_IF
    ELSE
      _nNctBaseUnitIdx              := 1;
      _nState                       := INIT_NCT_BASE_UNIT_ITF;

      IF (_eMessageLevel = E_MessageType.eMessageVerbose)
      THEN
        _stMsg.eType                := E_MessageType.eMessageVerbose;
        _stMsg.eSubdevice           := e_Subdevice.Xpu_fbNctBaseUnit;
        _stMsg.iErrorNumber         := _nNctBaseUnitCount;
        _stMsg.sText                := concat(TO_STRING(_eState), ': ');
        _stMsg.sText                := concat(_stMsg.sText, TO_STRING(_nState));
        f_MessageSet(_stMsg);
      END_IF
    END_IF

  //-----------------------------------------------------------------------------------------------
  //-----------------------------------------------------------------------------------------------
  INIT_NCT_BASE_UNIT_ITF:
    _ItfNctBaseUnit[_nNctBaseUnitIdx] := _fbNctController.BaseUnitInterfaceTcIo(_nNctBaseUnitIdx);
    _nState                           := INIT_NCT_BASE_UNIT_NEXT;

  //-----------------------------------------------------------------------------------------------
  //-----------------------------------------------------------------------------------------------
  INIT_NCT_BASE_UNIT_NEXT:
    IF (_nNctBaseUnitIdx > _nNctBaseUnitCount-1)
    THEN
      _eState                       := E_PROGRESS.PROGRESS_OCCUPIED;
    ELSE
      _nNctBaseUnitIdx              := _nNctBaseUnitIdx + 1;
      _nState                       := INIT_NCT_BASE_UNIT_ITF;
    END_IF
  END_CASE
END_CASE
//-----------------------------------------------------------------------------------------------
//-----------------------------------------------------------------------------------------------
//-----------------------------------------------------------------------------------------------
CASE _eState
OF
  E_PROGRESS.PROGRESS_OCCUPIED:     // reserve
    _eState                         := E_PROGRESS.PROGRESS_WORKING;
END_CASE
//-----------------------------------------------------------------------------------------------
//-----------------------------------------------------------------------------------------------
//-----------------------------------------------------------------------------------------------
CASE _eState
OF
  E_PROGRESS.PROGRESS_WORKING:      // reserve
    _eState                         := E_PROGRESS.PROGRESS_STILL_WORKING;
    _nState                         := INIT_TRACK_COM;
END_CASE
//-----------------------------------------------------------------------------------------------
//-----------------------------------------------------------------------------------------------
//-----------------------------------------------------------------------------------------------
CASE _eState
OF
  E_PROGRESS.PROGRESS_STILL_WORKING:// connect local instances of track, part, modules and mover
  CASE _nState
  OF
  //-----------------------------------------------------------------------------------------------
  //-----------------------------------------------------------------------------------------------
  INIT_TRACK_COM:                   // get TcCom Object for my track (_nTrack is fixed to 1 in this example; multi track is not intended)
    IF _fbXpuTrack.GetComObject(_Track_OTCID[_nTrack])
    THEN
      _nState                       := INIT_PART_COM;

      IF (_eMessageLevel = E_MessageType.eMessageVerbose)
      THEN
        _stMsg.eType                := E_MessageType.eMessageVerbose;
        _stMsg.eSubdevice           := e_Subdevice.Xpu_fbXpuTrack;
        _stMsg.iErrorNumber         := _nTrack;
        _stMsg.sText                := concat(TO_STRING(_eState), ': ');
        _stMsg.sText                := concat(_stMsg.sText, TO_STRING(_nState));
        f_MessageSet(_stMsg);
      END_IF
    END_IF
  //-----------------------------------------------------------------------------------------------
  //-----------------------------------------------------------------------------------------------
  INIT_PART_COM:                    // get TcCom object for my part (also fixed to 1 part per ProcessingUnit; multi part is not intended)
    IF _fbXpuPart.GetComObject(_Part_OTCID[1])
    THEN
      _nState                       := INIT_PART_MODULE_COUNT;

      IF (_eMessageLevel = E_MessageType.eMessageVerbose)
      THEN
        _stMsg.eType                := E_MessageType.eMessageVerbose;
        _stMsg.eSubdevice           := e_Subdevice.Xpu_fbXpuPart;
        _stMsg.iErrorNumber         := 1;
        _stMsg.sText                := concat(TO_STRING(_eState), ': ');
        _stMsg.sText                := concat(_stMsg.sText, TO_STRING(_nState));
        f_MessageSet(_stMsg);
      END_IF
    END_IF
  //-----------------------------------------------------------------------------------------------
  //-----------------------------------------------------------------------------------------------
  INIT_PART_MODULE_COUNT:           // get count of motor modules
    _nModuleCount                   := TO_UINT(_fbXpuPart.GetModuleCount());
  
    IF (_nModuleCount > 0)          // one is enough
    THEN
      _nState                       := INIT_PART_MODULE_OID;

      IF (_eMessageLevel = E_MessageType.eMessageVerbose)
      THEN
        _stMsg.eType                := E_MessageType.eMessageVerbose;
        _stMsg.eSubdevice           := e_Subdevice.Xpu_fbXpuPart;
        _stMsg.iErrorNumber         := _nModuleCount;
        _stMsg.sText                := concat(TO_STRING(_eState), ': ');
        _stMsg.sText                := concat(_stMsg.sText, TO_STRING(_nState));
        f_MessageSet(_stMsg);
      END_IF
    END_IF
  //-----------------------------------------------------------------------------------------------
  //-----------------------------------------------------------------------------------------------
  INIT_PART_MODULE_OID:             // get object IDs of all motor modules in part
    IF _fbXpuPart.GetModuleOids()
    THEN
      _Module_OTCID                 := _fbXpuPart.P_ModuleOids; // copy IDs to local
  
      _nState                       := INIT_PART_MODULE_COM;    // go, connect module IDs
      _nModuleIdx                   := 1;                       // start at first module

      IF (_eMessageLevel = E_MessageType.eMessageVerbose)
      THEN
        _stMsg.eType                := E_MessageType.eMessageVerbose;
        _stMsg.eSubdevice           := e_Subdevice.Xpu_fbPartModules;
        _stMsg.iErrorNumber         := _nModuleIdx;
        _stMsg.sText                := concat(TO_STRING(_eState), ': ');
        _stMsg.sText                := concat(_stMsg.sText, TO_STRING(_nState));
        //f_MessageSet(_stMsg);
      END_IF
    END_IF
  //-----------------------------------------------------------------------------------------------
  //-----------------------------------------------------------------------------------------------
  INIT_PART_MODULE_COM:           // connect to TcCom object
    IF _fbPartModules[_nModuleIdx].GetComObject(_Module_OTCID[_nModuleIdx])
    THEN
      _nState                       := INIT_PART_MODULE_COM_NEXT;
    END_IF
  //-----------------------------------------------------------------------------------------------
  INIT_PART_MODULE_COM_NEXT:
    IF (_nModuleIdx > _nModuleCount-1)
    THEN
      // all data from modules collected, continue to mover data
      _nState                       := INIT_MOVER_COM;          // go, connect mover IDs 
      _nMoverIdx                    :=  1;                      // start at first mover

      IF (_eMessageLevel = E_MessageType.eMessageVerbose)
      THEN
        _stMsg.eType                := E_MessageType.eMessageVerbose;
        _stMsg.eSubdevice           := e_Subdevice.Xpu_fbMoverXpu;
        _stMsg.iErrorNumber         := _nMoverIdx;
        _stMsg.sText                := concat(TO_STRING(_eState), ': ');
        _stMsg.sText                := concat(_stMsg.sText, TO_STRING(_nState));
        //f_MessageSet(_stMsg);
      END_IF
    ELSE
      // still data to fetch, increment search index, go back to fetching data
      _nState                       := INIT_PART_MODULE_COM;    // go back for next
      _nModuleIdx                   := _nModuleIdx + 1;       // next

      IF (_eMessageLevel = E_MessageType.eMessageVerbose)
      THEN
        _stMsg.eType                := E_MessageType.eMessageVerbose;
        _stMsg.eSubdevice           := e_Subdevice.Xpu_fbPartModules;
        _stMsg.iErrorNumber         := _nModuleIdx;
        _stMsg.sText                := concat(TO_STRING(_eState), ': ');
        _stMsg.sText                := concat(_stMsg.sText, TO_STRING(_nState));
        //f_MessageSet(_stMsg);
      END_IF
    END_IF
  //-----------------------------------------------------------------------------------------------
  //-----------------------------------------------------------------------------------------------
  INIT_MOVER_COM:                   // connect to TcCom object
    IF _fbMoverXpu[_nMoverIdx].GetComObject(_Mov_OTCID[_nMoverIdx])
    THEN
      _nState                       := INIT_MOVER_COM_NEXT;
    END_IF
  //-----------------------------------------------------------------------------------------------
  INIT_MOVER_COM_NEXT:
    IF (_nMoverIdx > _nMoverCount-1)
    THEN
      // all done
      _nState                       := INIT_DATA_GET;           // get important data from ProcessingUnit etc...

      IF (_eMessageLevel = E_MessageType.eMessageVerbose)
      THEN
        _stMsg.eType                := E_MessageType.eMessageVerbose;
        _stMsg.eSubdevice           := e_Subdevice.Xpu_fbProcessingUnit;
        _stMsg.iErrorNumber         := 0;
        _stMsg.sText                := concat(TO_STRING(_eState), ': ');
        _stMsg.sText                := concat(_stMsg.sText, TO_STRING(_nState));
        f_MessageSet(_stMsg);
      END_IF
    ELSE
      // more data to fetch, increment search index and go back
      _nState                       := INIT_MOVER_COM;          // go back for next
      _nMoverIdx                    := _nMoverIdx + 1;       // next

      IF (_eMessageLevel = E_MessageType.eMessageVerbose)
      THEN
        _stMsg.eType                := E_MessageType.eMessageVerbose;
        _stMsg.eSubdevice           := e_Subdevice.Xpu_fbMoverXpu;
        _stMsg.iErrorNumber         := _nMoverIdx;
        _stMsg.sText                := concat(TO_STRING(_eState), ': ');
        _stMsg.sText                := concat(_stMsg.sText, TO_STRING(_nState));
        //f_MessageSet(_stMsg);
      END_IF
    END_IF
  //-----------------------------------------------------------------------------------------------
  //-----------------------------------------------------------------------------------------------
  INIT_DATA_GET:                    // get data, add more if your application requires it
    // start counter
    _eDataGetCount                  := _eDataGetCount + 1;
    IF (_eDataGetCount MOD E_PROGRESS.PROGRESS_ERROR = 0)
    THEN
      _eState                       := E_PROGRESS.PROGRESS_ERROR;
      _eCheck                       := E_XPU_CHECK.PROCESSING_UNIT_GET_DATA_EXCEED;

      _stMsg.eType                  := E_MessageType.eMessageError;
      _stMsg.eSubdevice             := e_Subdevice.Xpu_fbProcessingUnit;
      _stMsg.iErrorNumber           := _nMoverIdx;
      _stMsg.sText                  := concat(TO_STRING(_nState), ': ');
      _stMsg.sText                  := concat(_stMsg.sText, TO_STRING(_eCheck));
      f_MessageSet(_stMsg);
    END_IF
    // wait for plausible data from members
    IF (_bAllPositionsValid) AND
       (_nLengthXpu > 0)
    THEN
      _nState                       := INIT_DATA_CHECK;
      _eChk                         := E_XPU_CHECK.PROCESSING_UNIT_POSITIONS_VALID;
      IF (_eMessageLevel > E_MessageType.eMessageError)
      THEN
        _stMsg.eType                := E_MessageType.eMessageInfo;
        _stMsg.eSubdevice           := e_Subdevice.Xpu_fbProcessingUnit;
        _stMsg.iErrorNumber         := 0;
        _stMsg.sText                := concat(TO_STRING(_nState), ': ');
        _stMsg.sText                := concat(_stMsg.sText, TO_STRING(E_XPU_CHECK.PROCESSING_UNIT_POSITIONS_VALID));
        f_MessageSet(_stMsg);
      END_IF
    END_IF

    _bAllPositionsValid             := _fbProcessingUnit.GetAreAllPositionsValid();
    _nDetectedMoverCount            := TO_UINT(_fbProcessingUnit.GetDetectedMoverCount());
    _nExpectedMoverCount            := TO_UINT(_fbProcessingUnit.GetExpectedMoverCount());

    _XpuOperationMode               := _fbProcessingUnit.GetOperationMode();
    _MoverIdDetectionMode           := _fbProcessingUnit.GetMoverIdDetectionMode();

    _RailLengthXpu                  := _fbXpuPart.GetLength();
    _RailLengthGroup                := _fbMc2CaGroup.GetRailLength();
    _nLengthXpu                     := TO_UINT(_RailLengthXpu);
    _nLengthGroup                   := TO_UINT(_RailLengthGroup);

  //-----------------------------------------------------------------------------------------------
  //-----------------------------------------------------------------------------------------------
  INIT_DATA_CHECK:                  // plausibility checks
    IF NOT (_nDetectedMoverCount = _nExpectedMoverCount)
    THEN
      _eChk                         := E_XPU_CHECK.MOVER_COUNT_NOT_EQUAL; // the thing that must not be
      _eState                       := E_PROGRESS.PROGRESS_ERROR;

      _stMsg.eType                  := E_MessageType.eMessageError;
      _stMsg.eSubdevice             := e_Subdevice.Xpu_fbProcessingUnit;
      _stMsg.iErrorNumber           := _nMoverIdx;
      _stMsg.sText                  := concat(TO_STRING(_nState), ': ');
      _stMsg.sText                  := concat(_stMsg.sText, TO_STRING(E_XPU_CHECK.MOVER_COUNT_NOT_EQUAL));
      f_MessageSet(_stMsg);

    ELSIF NOT (_nLengthXpu = _nLengthGroup)
    THEN
      _eChk                         := E_XPU_CHECK.RAIL_LENGTH_COMPARE;   // yet another thing that must not be
      _eState                       := E_PROGRESS.PROGRESS_ERROR;

      _stMsg.eType                  := E_MessageType.eMessageError;
      _stMsg.eSubdevice             := e_Subdevice.Xpu_fbProcessingUnit;
      _stMsg.iErrorNumber           := _nMoverIdx;
      _stMsg.sText                  := concat(TO_STRING(_nState), ': ');
      _stMsg.sText                  := concat(_stMsg.sText, TO_STRING(E_XPU_CHECK.RAIL_LENGTH_COMPARE));
      f_MessageSet(_stMsg);
    ELSE
      _sVersionXpu                  := _fbProcessingUnit.GetVersionString();
      _nState                       := INIT_DONE;                         // write success
    END_IF

  //-----------------------------------------------------------------------------------------------
  //-----------------------------------------------------------------------------------------------
  INIT_DONE:
    _eState                         := E_PROGRESS.PROGRESS_DONE;          // method is done
    IF (_eMessageLevel > E_MessageType.eMessageError)
    THEN
      _stMsg.eType                  := E_MessageType.eMessageInfo;
      _stMsg.eSubdevice             := e_Subdevice.Xpu_fbProcessingUnit;
      _stMsg.iErrorNumber           := 0;
      _stMsg.sText                  := concat('Xpu VersionString: ', _sVersionXpu);
      f_MessageSet(_stMsg);

      _stMsg.eType                  := E_MessageType.eMessageInfo;
      _stMsg.eSubdevice             := e_Subdevice.Xpu_fbProcessingUnit;
      _stMsg.iErrorNumber           := 0;
      _stMsg.sText                  := concat(TO_STRING(_nState), ': ');
      _stMsg.sText                  := concat(_stMsg.sText, TO_STRING(_eState));
      f_MessageSet(_stMsg);
    END_IF
  END_CASE
END_CASE
//-----------------------------------------------------------------------------------------------
//-----------------------------------------------------------------------------------------------
//-----------------------------------------------------------------------------------------------
_eReslt                             := _eState;
XpuInit                             := _nState;
//-----------------------------------------------------------------------------------------------
//-----------------------------------------------------------------------------------------------
//-----------------------------------------------------------------------------------------------
END_METHOD

PROPERTY XpuInstance : uint
SET
//
// Who am I?
// Environment may have more than one ProcessingUnit,
// information required for connecting to the correct instance of ProcessingUnit
_nXpu := XpuInstance;
END_SET
END_PROPERTY

PROPERTY XpuModuleInfoData : REFERENCE TO ARRAY[1..MAX_MODULE] OF Tc3_XTS_Utility.ST_InfoDataView
SET

_ModuleInfoData REF= XpuModuleInfoData;
END_SET
END_PROPERTY

PROPERTY XpuOtcid : OTCID
GET
XpuOtcid := _Xpu_OTCID;
END_GET
END_PROPERTY

END_FUNCTION_BLOCK

// ---- XTS/XtsTransportUnit/fb_TransportUnit.TcPOU
//---------------------------------------------------------------------------------------------------------------
//
//  HAUD 2024.03.18
//
//  - XTS_TRANSPORT_LAYER
//
//  fb_TransportUnit
//  - Ctrl/STate interface, reacts to change of command
//    - Cmd(E_TRANSPORT_CTRL)
//
//  - controls members via structures and interfaces for getting XTS in defined state
//    - CMD_INIT:
//        - XPU is initialized:         XTS_CMD_INIT + PROGRESS_DONE
//        - XPU cyclic checks enabled:  XTS_IDLE     + PROGRESS_WORKING
//        - XPU detects mover:          _XpuState.Check == MOVER_ID_DETECTION_VALID
//
//    - CMD_IDLE
//      - Cyclic Checks of XPU and CaGroup
//        - XPU cyclic checks enabled:  XTS_IDLE     + PROGRESS_WORKING
//
//
//  CTRL / STATE --> see proprerties
//  structs for use of function block via mapping
//  cyclic check for new command
//
//  VAR INPUT / OUTPUT --> see properties
//
//---------------------------------------------------------------------------------------------------------------
// This SOFTWARE is provided as an Exemple by THE PROVIDER "as is" and "with all faults." THE PROVIDER makes no 
// representations or warranties of any kind concerning the safety, suitability, lack of viruses, inaccuracies, 
// typographical errors, or other harmful components of this SOFTWARE. There are inherent dangers in the use of 
// any software, and you are solely responsible for determining whether this SOFTWARE is compatible with your 
// equipment and other software installed on your equipment. You are also solely responsible for the protection 
// of your equipment and backup of your data, and THE PROVIDER will not be liable for any damages you may suffer 
// in connection with using, modifying, or distributing this SOFTWARE.
//---------------------------------------------------------------------------------------------------------------
FUNCTION_BLOCK fb_TransportUnit
VAR
  _eCheck                       : E_XTS_TRANSPORT_CHECK;

  // Transport Ctrl/State
  _Ctrl                         : REFERENCE TO ST_XTS_TRANSPORT_CTRL;
  _State                        : REFERENCE TO ST_XTS_TRANSPORT_STATE;


  // execute transport commands
  _eCmd,
  _eCmdOld                      : E_XTS_TRANSPORT_CTRL;

  // execution state
  _eState                       : E_XTS_TRANSPORT_STATE;

  // execution result
  _eJobResult,
  _eResult                      : E_PROGRESS;


  // members of transport
  _XpuCtrl                      : REFERENCE TO ST_XPU_CTRL;                     // processing unit ctrl
  _XpuState                     : REFERENCE TO ST_XPU_STATE;                    // processing unit state
  _XpuInfo                      : REFERENCE TO ST_XPU_INFO;                     // processing unit information

  _GroupItf                     : I_XtsTransport_CaGroup;                       // group methods
  _GroupInfo                    : REFERENCE TO ST_GROUP_INFO;                   // info from group

  _MoverItf                     : REFERENCE TO ARRAY[1..MAX_MOVER] OF I_XtsTransport_Mover;   // mover methods
  _MoverInfo                    : REFERENCE TO ARRAY[1..MAX_MOVER] OF ST_MOVER_INFO;          // info from mover
  _MoverLastPosition            : REFERENCE TO ARRAY[1..MAX_MOVER] OF LREAL;                  // last commanded position of mover
  _MoverLastGap                 : REFERENCE TO ARRAY[1..MAX_MOVER] OF LREAL;                  // last commanded gapp of mover

  _StationStart                 : REFERENCE TO ST_STATION_PARAMETER;            // position, gap, dynamic constraints for sending all mover to start position

  // stations lists
  _ItfStationList               : REFERENCE TO ARRAY[1..MAX_STATION]  OF I_Station_LinkedList;  // access to all stations lists

  // station controls
  _StationControl               : REFERENCE TO ARRAY[1..MAX_STATION]  OF ST_STATION_CTRL;

  // station states
  _StationState                 : REFERENCE TO ARRAY[1..MAX_STATION]  OF ST_STATION_STATE;


  // access to stations methods by interface
  _ItfStationCtrl               : REFERENCE TO ARRAY[1..MAX_STATION]  OF I_XtsTransport_Station;

  _nStartStation                : UINT;

  _stMoverDataSend              : ST_STATION_MOVER_DATA;    // mover ticket data

  _stListResult                 : ST_STATION_LIST_RESULT;   // Xts station linkedlist entry

  _eMessageLevel                : E_MessageType;
  _stMsg                        : ST_Message;
END_VAR

IF NOT Check() THEN RETURN; END_IF

_stMsg.eDevice                  := XtsTransportUnit + 1;

_eCmd                           := _Ctrl.Cmd;
// check for command change
// get state for cmd
IF (_eCmd <> _eCmdOld)
THEN
  _eState                       := Cmd(_eCmd);
  _eCmdOld                      := _eCmd;

  IF (_eMessageLevel = E_MessageType.eMessageVerbose)
  THEN
    _stMsg.eType                := E_MessageType.eMessageVerbose;
    _stMsg.eSubdevice           := e_Subdevice.TransportUnit_General;
    _stMsg.iErrorNumber         := 0;
    _stMsg.sText                := concat( 'Command: ', TO_STRING(_eCmd));
    _stMsg.sText                := concat(_stMsg.sText, ': ');
    _stMsg.sText                := concat(_stMsg.sText, TO_STRING(_eResult));
    f_MessageSet(_stMsg);
  END_IF
END_IF

CASE _eResult
OF
  E_PROGRESS.PROGRESS_INVALID:
    _State.State                := TO_UINT(_eResult);

  E_PROGRESS.PROGRESS_ERROR:
    _State.State                := _eState + E_PROGRESS.PROGRESS_ERROR;

  E_PROGRESS.PROGRESS_DONE:
    _State.State                := _eState + E_PROGRESS.PROGRESS_DONE;

    IF (_GroupInfo.GroupErrorStop) OR
       (_GroupInfo.GroupError)     OR
       NOT (_XpuInfo.AllPositionsValid)
    THEN
      _eResult                  := E_PROGRESS.PROGRESS_ERROR;
    END_IF
ELSE
  _State.State                  := _eState + _eResult;

  CASE _eState
  OF
    E_XTS_TRANSPORT_STATE.TRANSPORT_INIT:
      _eResult                  := XpuInit(TRUE);
  
    E_XTS_TRANSPORT_STATE.TRANSPORT_IDLE:
      _eResult                  := f_GetProgress(_XpuState.State);
  
      IF (_GroupInfo.GroupErrorStop) OR
         (_GroupInfo.GroupError)     OR
         NOT (_XpuInfo.AllPositionsValid)
      THEN
        _eResult                := E_PROGRESS.PROGRESS_ERROR;
      END_IF
  
    E_XTS_TRANSPORT_STATE.TRANSPORT_MOVER_ENABLE:
      IF NOT (_XpuState.DcLink)
      THEN
        _eResult                := E_PROGRESS.PROGRESS_BUSY;

      ELSIF NOT (_XpuInfo.AllPositionsValid)
      THEN
        _eResult                := E_PROGRESS.PROGRESS_ERROR;
      ELSE
        _eResult                := MoverEnableAll(TRUE);
      END_IF
  
    E_XTS_TRANSPORT_STATE.TRANSPORT_MOVER_DISABLE:
      _eResult                  := MoverDisableAll(TRUE);

    E_XTS_TRANSPORT_STATE.TRANSPORT_MOVER_HALT_CA:
      _eResult                  := MoverHaltAll(TRUE);

    E_XTS_TRANSPORT_STATE.TRANSPORT_MOVER_STOP:
      _eResult                  := MoverStopAll(TRUE);
  
    E_XTS_TRANSPORT_STATE.TRANSPORT_GROUP_CLEAR:
      _eResult                  := GroupClear(TRUE);
  
    E_XTS_TRANSPORT_STATE.TRANSPORT_GROUP_BUILD:
      _eResult                  := GroupBuild(TRUE);
  
    E_XTS_TRANSPORT_STATE.TRANSPORT_GROUP_ENABLE:
      _eResult                  := GroupEnable(TRUE);

    E_XTS_TRANSPORT_STATE.TRANSPORT_GROUP_STOP:
      _eResult                  := GroupStop(TRUE);

    E_XTS_TRANSPORT_STATE.TRANSPORT_START:
      IF NOT (_XpuState.DcLink)
      THEN
        _eResult                := E_PROGRESS.PROGRESS_BUSY;

      ELSIF NOT (_XpuInfo.AllPositionsValid)
      THEN
        _eResult                := E_PROGRESS.PROGRESS_ERROR;
      ELSE
        _eResult                := TransportStart(TRUE);
      END_IF
  
    E_XTS_TRANSPORT_STATE.TRANSPORT_RESTART:
      IF NOT (_XpuState.DcLink)
      THEN
        _eResult                := E_PROGRESS.PROGRESS_BUSY;

      ELSIF NOT (_XpuInfo.AllPositionsValid)
      THEN
        _eResult                := E_PROGRESS.PROGRESS_ERROR;
      ELSE
        _eResult                := TransportRestart(TRUE);
      END_IF
  ELSE
    _eResult                    := E_PROGRESS.PROGRESS_INVALID;
  END_CASE

END_CASE

_State.XpuState                 := _XpuState;
_State.XpuInfo                  := _XpuInfo;
_State.GroupInfo                := _GroupInfo;

METHOD PRIVATE Check  : BOOL
VAR_INST
  _idx        : UINT;
END_VAR

IF NOT __ISVALIDREF(_Ctrl)
THEN
  _eCheck                     := E_XTS_TRANSPORT_CHECK.POINTER_NULL_CTRL;
  RETURN;
END_IF

IF NOT __ISVALIDREF(_State)
THEN
  _eCheck                     := E_XTS_TRANSPORT_CHECK.POINTER_NULL_STATE;
  RETURN;
END_IF

_State.Check                  := _eCheck;

IF NOT __ISVALIDREF(_XpuCtrl)
THEN
  _eCheck                     := E_XTS_TRANSPORT_CHECK.POINTER_NULL_XPU_CTRL;
  RETURN;
END_IF

IF NOT __ISVALIDREF(_XpuState)
THEN
  _eCheck                     := E_XTS_TRANSPORT_CHECK.POINTER_NULL_XPU_STATE;
  RETURN;
END_IF

IF NOT __ISVALIDREF(_XpuInfo)
THEN
  _eCheck                     := E_XTS_TRANSPORT_CHECK.POINTER_NULL_XPU_INFO;
  RETURN;
END_IF

IF NOT (_GroupItf <> 0)
THEN
  _eCheck                     := E_XTS_TRANSPORT_CHECK.POINTER_NULL_GROUP_ITF;
  RETURN;
END_IF

IF NOT __ISVALIDREF(_GroupInfo)
THEN
  _eCheck                     := E_XTS_TRANSPORT_CHECK.POINTER_NULL_GROUP_INFO;
  RETURN;
END_IF

IF NOT __ISVALIDREF(_MoverItf)
THEN
  _eCheck                     := E_XTS_TRANSPORT_CHECK.POINTER_NULL_MOVER;
  RETURN;
END_IF

FOR _idx := 1 TO MAX_MOVER
DO
  IF NOT (_MoverItf[_idx] <> 0)
  THEN
    _eCheck                   := E_XTS_TRANSPORT_CHECK.POINTER_NULL_MOVER_ITF;
    RETURN;
  END_IF
END_FOR

IF NOT __ISVALIDREF(_MoverInfo)
THEN
  _eCheck                     := E_XTS_TRANSPORT_CHECK.POINTER_NULL_MOVER_INFO;
  RETURN;
END_IF

IF NOT __ISVALIDREF(_MoverLastPosition)
THEN
  _eCheck                     := E_XTS_TRANSPORT_CHECK.POINTER_NULL_MOVER_LAST_POS;
  RETURN;
END_IF

IF NOT __ISVALIDREF(_MoverLastGap)
THEN
  _eCheck                     := E_XTS_TRANSPORT_CHECK.POINTER_NULL_MOVER_LAST_GAP;
  RETURN;
END_IF

IF NOT __ISVALIDREF(_StationStart)
THEN
  _eCheck                     := E_XTS_TRANSPORT_CHECK.POINTER_NULL_STATION_START;
  RETURN;
END_IF

IF NOT __ISVALIDREF(_ItfStationList)
THEN
  _eCheck                     := E_XTS_TRANSPORT_CHECK.POINTER_NULL_STATION_ITF;
  RETURN;
END_IF

IF NOT __ISVALIDREF(_StationControl)
THEN
  _eCheck                     := E_XTS_TRANSPORT_CHECK.POINTER_NULL_STATION_CONTROL;
  RETURN;
END_IF

IF NOT __ISVALIDREF(_StationState)
THEN
  _eCheck                     := E_XTS_TRANSPORT_CHECK.POINTER_NULL_STATION_STATE;
  RETURN;
END_IF

IF NOT __ISVALIDREF(_ItfStationCtrl)
THEN
  _eCheck                     := E_XTS_TRANSPORT_CHECK.POINTER_NULL_STATION_CTRL_ITF;
  RETURN;
END_IF


_eCheck                       := E_XTS_TRANSPORT_CHECK.DONE_CHECK;
Check                         := TRUE;
END_METHOD

METHOD PRIVATE Cmd : E_XTS_TRANSPORT_STATE
VAR_INPUT
  Ctrl      : E_XTS_TRANSPORT_CTRL;
END_VAR
VAR_INST
  _eState   : E_XTS_TRANSPORT_STATE;
END_VAR
IF NOT Check() THEN RETURN; END_IF


CASE Ctrl
OF
  E_XTS_TRANSPORT_CTRL.CMD_NULL:  // clear all method calls
    _eState               := E_XTS_TRANSPORT_STATE.TRANSPORT_NULL;
    _eResult              := XpuInit         (FALSE);
    _eResult              := GroupClear      (FALSE);
    _eResult              := GroupBuild      (FALSE);
    _eResult              := GroupEnable     (FALSE);
    _eResult              := GroupStop       (FALSE);
    _eResult              := MoverEnableAll  (FALSE);
    _eResult              := MoverDisableAll (FALSE);
    _eResult              := MoverHaltAll    (FALSE);
    _eResult              := MoverStopAll    (FALSE);
    _eResult              := TransportStart  (FALSE);
    _eResult              := TransportRestart(FALSE);

  E_XTS_TRANSPORT_CTRL.CMD_INIT:  // clear methods for initialization
    _eState               := E_XTS_TRANSPORT_STATE.TRANSPORT_INIT;
    _eResult              := XpuInit(FALSE);


ELSE
  IF NOT (_XpuState.Init = E_XPU_INIT.INIT_DONE)
  THEN
    // no init, no further commands possible
    _eState               := E_XTS_TRANSPORT_STATE.TRANSPORT_INVALID;
  ELSE
    CASE Ctrl
    OF
      E_XTS_TRANSPORT_CTRL.CMD_IDLE:
        _eState           := E_XTS_TRANSPORT_STATE.TRANSPORT_IDLE;

      E_XTS_TRANSPORT_CTRL.CMD_MOVER_ENABLE:
        _eState           := E_XTS_TRANSPORT_STATE.TRANSPORT_MOVER_ENABLE;
        _eResult          := MoverEnableAll(FALSE);

      E_XTS_TRANSPORT_CTRL.CMD_MOVER_DISABLE:
        _eState           := E_XTS_TRANSPORT_STATE.TRANSPORT_MOVER_DISABLE;
        _eResult          := MoverDisableAll(FALSE);

      E_XTS_TRANSPORT_CTRL.CMD_MOVER_HALT_CA:
        _eState           := E_XTS_TRANSPORT_STATE.TRANSPORT_MOVER_HALT_CA;
        _eResult          := MoverHaltAll(FALSE);

      E_XTS_TRANSPORT_CTRL.CMD_MOVER_STOP:
        _eState           := E_XTS_TRANSPORT_STATE.TRANSPORT_MOVER_STOP;
        _eResult          := MoverStopAll(FALSE);

      E_XTS_TRANSPORT_CTRL.CMD_GROUP_CLEAR:
        _eState           := E_XTS_TRANSPORT_STATE.TRANSPORT_GROUP_CLEAR;
        _eResult          := GroupClear (FALSE);

      E_XTS_TRANSPORT_CTRL.CMD_GROUP_BUILD:
        _eState           := E_XTS_TRANSPORT_STATE.TRANSPORT_GROUP_BUILD;
        _eResult          := GroupBuild (FALSE);

      E_XTS_TRANSPORT_CTRL.CMD_GROUP_ENABLE:
        _eState           := E_XTS_TRANSPORT_STATE.TRANSPORT_GROUP_ENABLE;
        _eResult          := GroupEnable(FALSE);

      E_XTS_TRANSPORT_CTRL.CMD_GROUP_STOP:
        _eState           := E_XTS_TRANSPORT_STATE.TRANSPORT_GROUP_STOP;
        _eResult          := GroupStop(FALSE);

      E_XTS_TRANSPORT_CTRL.CMD_TRANSPORT_START:
        _eState           := E_XTS_TRANSPORT_STATE.TRANSPORT_START;
        _eResult          := TransportStart(FALSE);

      E_XTS_TRANSPORT_CTRL.CMD_TRANSPORT_RESTART:
        _eState           := E_XTS_TRANSPORT_STATE.TRANSPORT_RESTART;
        _eResult          := TransportRestart(FALSE);

    ELSE
        _eState           := E_XTS_TRANSPORT_STATE.TRANSPORT_INVALID;
    END_CASE
  END_IF
END_CASE

Cmd                       := _eState;
END_METHOD

PROPERTY Ctrl : REFERENCE TO ST_XTS_TRANSPORT_CTRL
SET
_Ctrl REF= Ctrl;
END_SET
END_PROPERTY

METHOD GroupBuild : E_PROGRESS
VAR_INPUT
  Execute     : BOOL;
END_VAR
VAR_INST
  _nErrorId   : UDINT;
  _eJobReslt,
  _eState     : E_PROGRESS;
END_VAR
//-----------------------------------------------------------------------------
IF NOT Execute 
THEN 
	_eState                       := E_PROGRESS.PROGRESS_INIT; 
END_IF 
//-----------------------------------------------------------------------------
IF NOT Check() 
THEN 
	GroupBuild                    := E_PROGRESS.PROGRESS_ERROR; 
	RETURN; 
END_IF
//-----------------------------------------------------------------------------
//-----------------------------------------------------------------------------
CASE _eState
OF
  E_PROGRESS.PROGRESS_INIT:
    IF Execute
    THEN
      _nErrorId                 := 0;

      IF (_GroupInfo.AxisCount <> 0)
      THEN
        _nErrorId               := 9999;
        _eState                 := E_PROGRESS.PROGRESS_ERROR;
      ELSE
        _eState                 := E_PROGRESS.PROGRESS_BUSY;
        _eJobReslt              := _GroupItf.AddAll(FALSE);
      END_IF
    END_IF
END_CASE
//---------------------------------------------------------------------------
//---------------------------------------------------------------------------
CASE _eState
OF
  E_PROGRESS.PROGRESS_BUSY:
    _eJobReslt                  := _GroupItf.AddAll(TRUE);

    IF (_eJobReslt = E_PROGRESS.PROGRESS_ERROR)
    THEN
      _eState                   := E_PROGRESS.PROGRESS_ERROR;

      _nErrorId                 := _GroupInfo.GroupErrorId;
      _eJobReslt                := _GroupItf.AddAll(FALSE);

    ELSIF (_eJobReslt = E_PROGRESS.PROGRESS_DONE)
    THEN
      _eState                   := E_PROGRESS.PROGRESS_PREPARE;
      _eJobReslt                := _GroupItf.AddAll(FALSE);
	  _eJobReslt				:= _GroupItf.Reset(FALSE);
    END_IF
END_CASE
//-----------------------------------------------------------------------------
//-----------------------------------------------------------------------------
CASE _eState
OF
  E_PROGRESS.PROGRESS_PREPARE:
    _eJobReslt                  := _GroupItf.Reset(TRUE);

    IF (_eJobReslt = E_PROGRESS.PROGRESS_ERROR)
    THEN
      _eState                   := E_PROGRESS.PROGRESS_ERROR;

      _nErrorId                 := _GroupInfo.GroupErrorId;
	    _eJobReslt				        := _GroupItf.Reset(FALSE);

    ELSIF (_eJobReslt = E_PROGRESS.PROGRESS_DONE)
    THEN
      _eState                   := E_PROGRESS.PROGRESS_DONE;
	    _eJobReslt				        := _GroupItf.Reset(FALSE);

      IF (_eMessageLevel = E_MessageType.eMessageVerbose)
      THEN
        _stMsg.eType            := E_MessageType.eMessageVerbose;
        _stMsg.eSubdevice       := e_Subdevice.TransportUnit_General;
        _stMsg.iErrorNumber     := 0;
        _stMsg.sText            := concat( 'State: ', TO_STRING(THIS^._eState));
        _stMsg.sText            := concat(_stMsg.sText, ': ');
        _stMsg.sText            := concat(_stMsg.sText, TO_STRING(_eState));
        f_MessageSet(_stMsg);
      END_IF
    END_IF
END_CASE
//-----------------------------------------------------------------------------
//-----------------------------------------------------------------------------

GroupBuild                      := _eState;
END_METHOD

METHOD GroupClear : E_PROGRESS
VAR_INPUT
  Execute     : BOOL;
END_VAR
VAR_INST
  _nRepeat,
  _nStation,
  _nErrorId   : UDINT;
  _eJobReslt,
  _eState     : E_PROGRESS;
END_VAR
//-----------------------------------------------------------------------------
IF NOT Execute 
THEN 
	_eState                       := E_PROGRESS.PROGRESS_INIT; 
END_IF 
//-----------------------------------------------------------------------------
IF NOT Check() 
THEN 
	GroupClear                    := E_PROGRESS.PROGRESS_ERROR; 
	RETURN; 
END_IF
//-----------------------------------------------------------------------------
//-----------------------------------------------------------------------------
CASE _eState
OF
  E_PROGRESS.PROGRESS_INIT:
    IF Execute
    THEN
      _nRepeat                  :=
      _nErrorId                 := 0;
      _eJobReslt                := _GroupItf.McHaltAll(FALSE);
      _eJobReslt                := _GroupItf.RemoveAll(FALSE);
      _eJobReslt                := _GroupItf.McResetAll(FALSE);
      _eJobReslt                := _GroupItf.Disable(FALSE);
      _eJobReslt                := _GroupItf.Reset(FALSE);
      _eJobReslt                := StationsClearOutfeed(FALSE);

      _eState                   := E_PROGRESS.PROGRESS_BUSY;
    END_IF
END_CASE
//---------------------------------------------------------------------------
//---------------------------------------------------------------------------
CASE _eState
OF
  E_PROGRESS.PROGRESS_BUSY:
    _eJobReslt                  := StationsClearOutfeed(TRUE);

    IF (_eJobReslt = E_PROGRESS.PROGRESS_DONE)
    THEN
      _eState                   := E_PROGRESS.PROGRESS_PREPARE;
      _eJobReslt                := StationsClearOutfeed(FALSE);
    END_IF

  //---------------------------------------------------------------------------
  //---------------------------------------------------------------------------
  E_PROGRESS.PROGRESS_PREPARE:
    _eJobReslt                  := _GroupItf.McHaltAll(TRUE);

    IF (_eJobReslt > E_PROGRESS.PROGRESS_STILL_WORKING)
    THEN
      _eState                   := E_PROGRESS.PROGRESS_STARTUP;
      _nErrorId                 := _GroupInfo.GroupErrorId;
      _eJobReslt                := _GroupItf.McHaltAll(FALSE);
    END_IF
  //---------------------------------------------------------------------------
  //---------------------------------------------------------------------------
  E_PROGRESS.PROGRESS_STARTUP:
    _eJobReslt                  := _GroupItf.RemoveAll(TRUE);

    IF (_eJobReslt > E_PROGRESS.PROGRESS_STILL_WORKING)
    THEN
      _eState                   := E_PROGRESS.PROGRESS_CHECK;
      _nErrorId                 := _GroupInfo.GroupErrorId;
      _eJobReslt                := _GroupItf.RemoveAll(FALSE);
    END_IF
  //---------------------------------------------------------------------------
  //---------------------------------------------------------------------------
  E_PROGRESS.PROGRESS_CHECK:
    _eJobReslt                  := _GroupItf.Disable(TRUE);

    IF (_eJobReslt > E_PROGRESS.PROGRESS_STILL_WORKING)
    THEN
      _eState                   := E_PROGRESS.PROGRESS_OCCUPIED;
      _nErrorId                 := _GroupInfo.GroupErrorId;
      _eJobReslt                := _GroupItf.Disable(FALSE);
    END_IF
  //---------------------------------------------------------------------------
  //---------------------------------------------------------------------------
  E_PROGRESS.PROGRESS_OCCUPIED:
    _eJobReslt                  := _GroupItf.Reset(TRUE);

    IF (_eJobReslt > E_PROGRESS.PROGRESS_STILL_WORKING)
    THEN
      _eState                   := E_PROGRESS.PROGRESS_WORKING;
      _nErrorId                 := _GroupInfo.GroupErrorId;
      _eJobReslt                := _GroupItf.Reset(FALSE);
    END_IF
END_CASE
//-----------------------------------------------------------------------------
//-----------------------------------------------------------------------------
CASE _eState
OF
  E_PROGRESS.PROGRESS_WORKING:
    IF    (_GroupInfo.AxisCount     = 0) AND
          (_GroupInfo.CaGroupState  = E_CA_GROUP_STATE.mcGroupStateDisabled) AND 
      NOT (_GroupInfo.GroupError)
    THEN
      _eState                   := E_PROGRESS.PROGRESS_DONE;

      IF (_eMessageLevel = E_MessageType.eMessageVerbose)
      THEN
        _stMsg.eType            := E_MessageType.eMessageVerbose;
        _stMsg.eSubdevice       := e_Subdevice.TransportUnit_General;
        _stMsg.iErrorNumber     := 0;
        _stMsg.sText            := concat( 'State: ', TO_STRING(THIS^._eState));
        _stMsg.sText            := concat(_stMsg.sText, ': ');
        _stMsg.sText            := concat(_stMsg.sText, TO_STRING(_eState));
        f_MessageSet(_stMsg);
      END_IF
    ELSE
      _nRepeat                  := _nRepeat + 1;
      IF NOT (_nRepeat > 2)
      THEN
        _eState                 := E_PROGRESS.PROGRESS_BUSY;
      ELSE
        _eState                 := E_PROGRESS.PROGRESS_ERROR;
      END_IF
    END_IF
END_CASE
//-----------------------------------------------------------------------------
//-----------------------------------------------------------------------------

GroupClear                      := _eState;
END_METHOD

METHOD GroupEnable : E_PROGRESS
VAR_INPUT
  Execute     : BOOL;
END_VAR
VAR_INST
  _nErrorId   : UDINT;
  _eJobReslt,
  _eState     : E_PROGRESS;
END_VAR
//-----------------------------------------------------------------------------
IF NOT Execute 
THEN 
	_eState                       := E_PROGRESS.PROGRESS_INIT; 
END_IF 
//-----------------------------------------------------------------------------
IF NOT Check() 
THEN 
	GroupEnable                   := E_PROGRESS.PROGRESS_ERROR; 
	RETURN; 
END_IF
//-----------------------------------------------------------------------------
//-----------------------------------------------------------------------------
CASE _eState
OF
  E_PROGRESS.PROGRESS_INIT:
    IF Execute
    THEN
      _nErrorId                 := 0;

      IF NOT (_GroupInfo.AxisCount <> 0)
      THEN
        _nErrorId               := 9999;
        _eState                 := E_PROGRESS.PROGRESS_ERROR;
      ELSE
        _eState                 := E_PROGRESS.PROGRESS_BUSY;
        _eJobReslt              := _GroupItf.Enable(FALSE);
      END_IF
    END_IF
END_CASE
//---------------------------------------------------------------------------
//---------------------------------------------------------------------------
CASE _eState
OF
  E_PROGRESS.PROGRESS_BUSY:
    _eJobReslt                  := _GroupItf.Enable(TRUE);

    IF (_eJobReslt = E_PROGRESS.PROGRESS_ERROR)
    THEN
      _eState                   := E_PROGRESS.PROGRESS_ERROR;

      _nErrorId                 := _GroupInfo.GroupErrorId;
      _eJobReslt                := _GroupItf.Enable(FALSE);

    ELSIF (_eJobReslt = E_PROGRESS.PROGRESS_DONE)
    THEN
      _eState                   := E_PROGRESS.PROGRESS_CHECK;
      _eJobReslt                := _GroupItf.Enable(FALSE);
    END_IF
END_CASE
//-----------------------------------------------------------------------------
//-----------------------------------------------------------------------------
CASE _eState
OF
  E_PROGRESS.PROGRESS_CHECK:
    IF (_GroupInfo.GroupStandby) OR
       (_GroupInfo.GroupMoving)  OR
       (_GroupInfo.GroupNotReady)
    THEN
      _eState                   := E_PROGRESS.PROGRESS_DONE;

      IF (_eMessageLevel = E_MessageType.eMessageVerbose)
      THEN
        _stMsg.eType            := E_MessageType.eMessageVerbose;
        _stMsg.eSubdevice       := e_Subdevice.TransportUnit_General;
        _stMsg.iErrorNumber     := 0;
        _stMsg.sText            := concat( 'State: ', TO_STRING(THIS^._eState));
        _stMsg.sText            := concat(_stMsg.sText, ': ');
        _stMsg.sText            := concat(_stMsg.sText, TO_STRING(_eState));
        f_MessageSet(_stMsg);
      END_IF
    ELSE
      IF (_GroupInfo.GroupErrorStop) OR
         (_GroupInfo.GroupError)
      THEN
        _eState                 := E_PROGRESS.PROGRESS_ERROR;
      END_IF
    END_IF
END_CASE
//-----------------------------------------------------------------------------
//-----------------------------------------------------------------------------
GroupEnable                     := _eState;
END_METHOD

PROPERTY GroupInfo : REFERENCE TO ST_GROUP_INFO
SET
_GroupInfo REF= GroupInfo;
END_SET
END_PROPERTY

PROPERTY GroupItf : I_XtsTransport_CaGroup
SET
_GroupItf := GroupItf;
END_SET
END_PROPERTY

METHOD GroupStop : E_PROGRESS
VAR_INPUT
  Execute     : BOOL;
END_VAR
VAR_INST
  _nRepeat,
  _nStation,
  _nErrorId   : UDINT;
  _eJobReslt,
  _eState     : E_PROGRESS;
END_VAR
//-----------------------------------------------------------------------------
IF NOT Execute 
THEN 
	_eState                      := E_PROGRESS.PROGRESS_INIT; 
END_IF 
//-----------------------------------------------------------------------------
IF NOT Check() 
THEN 
	GroupStop                    := E_PROGRESS.PROGRESS_ERROR; 
	RETURN; 
END_IF
//-----------------------------------------------------------------------------
//-----------------------------------------------------------------------------
CASE _eState
OF
  E_PROGRESS.PROGRESS_INIT:
    IF Execute
    THEN
      _nRepeat                  :=
      _nErrorId                 := 0;
      _eJobReslt                := _GroupItf.Stop(FALSE);

      _eState                   := E_PROGRESS.PROGRESS_BUSY;
    END_IF
END_CASE
//---------------------------------------------------------------------------
//---------------------------------------------------------------------------
CASE _eState
OF
  E_PROGRESS.PROGRESS_BUSY:
    _eJobReslt                  := _GroupItf.Stop(TRUE);

    IF (_eJobReslt = E_PROGRESS.PROGRESS_ERROR)
    THEN
      _eState                   := E_PROGRESS.PROGRESS_PREPARE;
      _nErrorId                 := _GroupInfo.GroupErrorId;
      _eJobReslt                := _GroupItf.Stop(FALSE);

    ELSIF (_eJobReslt = E_PROGRESS.PROGRESS_DONE)
    THEN
      _eState                   := E_PROGRESS.PROGRESS_WORKING;
      _eJobReslt                := _GroupItf.Stop(FALSE);
    END_IF
END_CASE
//-----------------------------------------------------------------------------
//-----------------------------------------------------------------------------
CASE _eState
OF
  E_PROGRESS.PROGRESS_WORKING:
    IF NOT (_GroupInfo.GroupError)
    THEN
      _eState                   := E_PROGRESS.PROGRESS_DONE;

      IF (_eMessageLevel = E_MessageType.eMessageVerbose)
      THEN
        _stMsg.eType            := E_MessageType.eMessageVerbose;
        _stMsg.eSubdevice       := e_Subdevice.TransportUnit_General;
        _stMsg.iErrorNumber     := 0;
        _stMsg.sText            := concat( 'State: ', TO_STRING(THIS^._eState));
        _stMsg.sText            := concat(_stMsg.sText, ': ');
        _stMsg.sText            := concat(_stMsg.sText, TO_STRING(_eState));
        f_MessageSet(_stMsg);
      END_IF
    ELSE
      IF (_GroupInfo.GroupErrorStop) OR
         (_GroupInfo.GroupError)
      THEN
        _nRepeat                := _nRepeat + 1;
        IF NOT (_nRepeat > 2)
        THEN
          _eState               := E_PROGRESS.PROGRESS_BUSY;
        ELSE
          _eState               := E_PROGRESS.PROGRESS_ERROR;
        END_IF
      END_IF
    END_IF
END_CASE
//-----------------------------------------------------------------------------
//-----------------------------------------------------------------------------

GroupStop                       := _eState;
END_METHOD

PROPERTY MessageLevel : e_messagetype
SET
_eMessageLevel := MessageLevel;
END_SET
END_PROPERTY

